C09153=1117.834,-111.203,-46.268,179.703,4.253,148.782
C09154=1117.839,-111.453,-46.260,179.703,4.248,148.781
C09155=1117.844,-111.703,-46.251,179.703,4.243,148.779
C09156=1117.850,-111.953,-46.242,179.703,4.238,148.778
C09157=1117.855,-112.203,-46.234,179.704,4.233,148.777
C09158=1117.861,-112.452,-46.225,179.705,4.228,148.776
C09159=1117.866,-112.702,-46.216,179.705,4.223,148.775
C09160=1117.872,-112.952,-46.207,179.705,4.218,148.773
C09161=1117.877,-113.202,-46.198,179.705,4.213,148.772
C09162=1117.881,-113.417,-46.191,179.706,4.208,148.771
C09163=1117.886,-113.632,-46.183,179.706,4.204,148.770
C09164=1117.890,-113.848,-46.175,179.706,4.199,148.769
C09165=1117.895,-114.063,-46.168,179.706,4.195,148.768
C09166=1117.900,-114.279,-46.161,179.706,4.190,148.767
C09167=1117.905,-114.494,-46.153,179.707,4.186,148.766
C09168=1117.909,-114.710,-46.145,179.707,4.181,148.765
C09169=1117.914,-114.925,-46.137,179.707,4.177,148.764
C09170=1117.919,-115.174,-46.129,179.707,4.171,148.763
C09171=1117.925,-115.424,-46.120,179.708,4.166,148.761
C09172=1117.930,-115.674,-46.112,179.708,4.161,148.760
C09173=1117.936,-115.924,-46.103,179.708,4.156,148.759
C09174=1117.941,-116.174,-46.094,179.709,4.150,148.757
C09175=1117.946,-116.423,-46.086,179.709,4.145,148.756
C09176=1117.952,-116.673,-46.077,179.709,4.139,148.755
C09177=1117.957,-116.923,-46.068,179.709,4.134,148.754
C09178=1117.962,-117.173,-46.060,179.709,4.129,148.753
C09179=1117.968,-117.422,-46.051,179.710,4.124,148.751
C09180=1117.973,-117.672,-46.042,179.710,4.119,148.750
C09181=1117.979,-117.923,-46.034,179.710,4.113,148.749
C09182=1117.984,-118.172,-46.025,179.711,4.108,148.748
C09183=1117.990,-118.422,-46.016,179.711,4.103,148.747
C09184=1117.995,-118.671,-46.008,179.712,4.098,148.745
C09185=1117.999,-118.922,-46.000,179.712,4.092,148.744
C09186=1118.005,-119.171,-45.991,179.712,4.087,148.743
C09187=1118.010,-119.421,-45.983,179.712,4.081,148.742
C09188=1118.016,-119.671,-45.974,179.712,4.076,148.740
C09189=1118.022,-119.920,-45.966,179.712,4.071,148.739
C09190=1118.027,-120.170,-45.957,179.713,4.066,148.738
C09191=1118.032,-120.420,-45.948,179.714,4.060,148.736
C09192=1118.038,-120.670,-45.940,179.714,4.055,148.735
C09193=1118.043,-120.920,-45.931,179.714,4.050,148.734
C09194=1118.049,-121.170,-45.923,179.714,4.045,148.733
C09195=1118.054,-121.419,-45.915,179.714,4.039,148.732
C09196=1118.059,-121.669,-45.906,179.714,4.033,148.730
C09197=1118.064,-121.919,-45.898,179.715,4.028,148.729
C09198=1118.070,-122.168,-45.890,179.715,4.023,148.728
C09199=1118.075,-122.418,-45.881,179.716,4.018,148.727
C09200=1118.081,-122.669,-45.873,179.715,4.012,148.725
C09201=1118.087,-122.918,-45.864,179.716,4.006,148.724
C09202=1118.091,-123.168,-45.856,179.717,4.001,148.723
C09203=1118.097,-123.417,-45.848,179.717,3.996,148.721
C09204=1118.103,-123.668,-45.840,179.717,3.991,148.720
C09205=1118.108,-123.917,-45.831,179.717,3.985,148.719
C09206=1118.114,-124.167,-45.823,179.717,3.979,148.718
C09207=1118.118,-124.417,-45.815,179.718,3.974,148.716
C09208=1118.123,-124.667,-45.806,179.718,3.969,148.715
C09209=1118.129,-124.916,-45.798,179.719,3.963,148.714
C09210=1118.135,-125.166,-45.789,179.718,3.957,148.713
C09211=1118.141,-125.416,-45.781,179.719,3.952,148.711
C09212=1118.145,-125.666,-45.773,179.719,3.947,148.710
C09213=1118.151,-125.915,-45.765,179.720,3.942,148.709
C09214=1118.157,-126.166,-45.757,179.720,3.935,148.707
C09215=1118.162,-126.416,-45.748,179.720,3.930,148.706
C09216=1118.167,-126.665,-45.741,179.721,3.925,148.705
C09217=1118.172,-126.915,-45.732,179.721,3.920,148.704
C09218=1118.177,-127.131,-45.725,179.721,3.914,148.702
C09219=1118.182,-127.345,-45.718,179.721,3.909,148.701
C09220=1118.187,-127.561,-45.711,179.721,3.905,148.700
C09221=1118.191,-127.776,-45.704,179.722,3.900,148.699
C09222=1118.196,-127.992,-45.697,179.722,3.895,148.698
C09223=1118.201,-128.207,-45.690,179.722,3.890,148.697
C09224=1118.205,-128.422,-45.683,179.723,3.886,148.696
C09225=1118.210,-128.639,-45.676,179.723,3.881,148.695
C09226=1117.787,-128.629,-45.702,179.730,3.886,148.693
C09227=1117.782,-128.414,-45.709,179.730,3.890,148.694
C09228=1117.777,-128.198,-45.716,179.729,3.895,148.696
C09229=1117.773,-127.982,-45.724,179.730,3.900,148.697
C09230=1117.768,-127.767,-45.730,179.729,3.904,148.698
C09231=1117.764,-127.551,-45.737,179.729,3.909,148.699
C09232=1117.759,-127.336,-45.744,179.729,3.914,148.700
C09233=1117.754,-127.120,-45.751,179.728,3.918,148.701
C09234=1117.750,-126.906,-45.758,179.728,3.923,148.702
C09235=1117.744,-126.655,-45.766,179.727,3.929,148.704
C09236=1117.738,-126.406,-45.775,179.728,3.935,148.705
C09237=1117.734,-126.156,-45.783,179.727,3.940,148.706
C09238=1117.728,-125.907,-45.791,179.727,3.945,148.707
C09239=1117.722,-125.656,-45.799,179.726,3.951,148.709
C09240=1117.717,-125.406,-45.808,179.726,3.957,148.710
C09241=1117.711,-125.157,-45.816,179.726,3.962,148.711
C09242=1117.707,-124.907,-45.824,179.726,3.967,148.712
C09243=1117.701,-124.657,-45.832,179.725,3.972,148.714
C09244=1117.696,-124.408,-45.841,179.725,3.978,148.715
C09245=1117.690,-124.158,-45.850,179.725,3.984,148.716
C09246=1117.684,-123.908,-45.858,179.725,3.989,148.717
C09247=1117.680,-123.658,-45.866,179.724,3.994,148.719
C09248=1117.674,-123.408,-45.874,179.724,3.999,148.720
C09249=1117.669,-123.159,-45.883,179.724,4.005,148.721
C09250=1117.663,-122.908,-45.891,179.724,4.011,148.723
C09251=1117.657,-122.659,-45.899,179.723,4.016,148.724
C09252=1117.652,-122.409,-45.908,179.722,4.021,148.725
C09253=1117.647,-122.159,-45.917,179.722,4.027,148.726
C09254=1117.642,-121.910,-45.924,179.722,4.032,148.728
C09255=1117.637,-121.660,-45.933,179.722,4.038,148.729
C09256=1117.631,-121.410,-45.942,179.721,4.043,148.730
C09257=1117.625,-121.160,-45.950,179.721,4.048,148.732
C09258=1117.620,-120.911,-45.959,179.721,4.054,148.733
C09259=1117.615,-120.660,-45.967,179.720,4.059,148.734
C09260=1117.610,-120.410,-45.976,179.720,4.064,148.735
C09261=1117.604,-120.161,-45.985,179.720,4.069,148.736
C09262=1117.598,-119.911,-45.993,179.720,4.075,148.738
C09263=1117.593,-119.661,-46.002,179.719,4.081,148.739
C09264=1117.588,-119.412,-46.010,179.719,4.086,148.740
C09265=1117.583,-119.162,-46.018,179.719,4.091,148.741
C09266=1117.577,-118.912,-46.027,179.719,4.096,148.743
C09267=1117.572,-118.663,-46.035,179.718,4.101,148.744
C09268=1117.567,-118.413,-46.044,179.718,4.107,148.745
C09269=1117.561,-118.162,-46.052,179.717,4.112,148.747
C09270=1117.556,-117.912,-46.061,179.717,4.117,148.748
C09271=1117.550,-117.663,-46.070,179.717,4.123,148.749
C09272=1117.545,-117.413,-46.079,179.717,4.128,148.750
C09273=1117.540,-117.164,-46.088,179.717,4.134,148.751
C09274=1117.534,-116.913,-46.096,179.716,4.139,148.753
C09275=1117.529,-116.664,-46.104,179.716,4.144,148.754
C09276=1117.523,-116.414,-46.113,179.716,4.149,148.755
C09277=1117.518,-116.164,-46.122,179.716,4.154,148.756
C09278=1117.513,-115.914,-46.131,179.715,4.159,148.757
C09279=1117.507,-115.665,-46.139,179.715,4.165,148.759
C09280=1117.502,-115.415,-46.148,179.714,4.170,148.760
C09281=1117.497,-115.165,-46.157,179.714,4.175,148.761
C09282=1117.491,-114.915,-46.165,179.714,4.180,148.763
C09283=1117.487,-114.700,-46.173,179.714,4.185,148.763
C09284=1117.482,-114.485,-46.181,179.713,4.190,148.765
C09285=1117.477,-114.270,-46.188,179.713,4.194,148.766
C09286=1117.473,-114.054,-46.196,179.713,4.198,148.767
C09287=1117.468,-113.838,-46.203,179.712,4.203,148.768
C09288=1117.463,-113.623,-46.211,179.713,4.207,148.769
C09289=1117.458,-113.408,-46.218,179.712,4.211,148.770
C09290=1117.454,-113.192,-46.226,179.712,4.217,148.771
C09291=1117.448,-112.943,-46.235,179.712,4.222,148.772
C09292=1117.443,-112.693,-46.244,179.711,4.227,148.773
C09293=1117.438,-112.443,-46.253,179.711,4.232,148.775
C09294=1117.433,-112.194,-46.262,179.711,4.237,148.776
C09295=1117.427,-111.944,-46.270,179.711,4.242,148.777
C09296=1117.422,-111.695,-46.279,179.710,4.248,148.778
C09297=1117.416,-111.445,-46.288,179.710,4.253,148.779
C09298=1117.411,-111.195,-46.297,179.710,4.258,148.781
C09299=1117.405,-110.945,-46.306,179.710,4.263,148.782
C09300=1117.400,-110.695,-46.315,179.709,4.267,148.783
C09301=1117.395,-110.445,-46.324,179.709,4.273,148.784
C09302=1117.390,-110.195,-46.333,179.708,4.278,148.785
C09303=1117.384,-109.946,-46.342,179.708,4.283,148.787
C09304=1117.379,-109.696,-46.350,179.708,4.288,148.788
C09305=1117.374,-109.446,-46.359,179.708,4.293,148.789
C09306=1117.368,-109.196,-46.369,179.707,4.298,148.790
C09307=1117.363,-108.946,-46.378,179.707,4.304,148.791
C09308=1117.358,-108.696,-46.387,179.707,4.309,148.793
C09309=1117.352,-108.447,-46.396,179.707,4.314,148.794
C09310=1117.347,-108.197,-46.404,179.706,4.319,148.795
C09311=1117.341,-107.947,-46.414,179.706,4.324,148.796
C09312=1117.336,-107.698,-46.423,179.706,4.329,148.797
C09313=1117.331,-107.448,-46.432,179.705,4.334,148.799
C09314=1117.326,-107.198,-46.441,179.705,4.339,148.800
C09315=1117.320,-106.948,-46.450,179.704,4.344,148.801
C09316=1117.314,-106.698,-46.459,179.704,4.349,148.802
C09317=1117.309,-106.448,-46.468,179.704,4.354,148.803
C09318=1117.304,-106.199,-46.477,179.704,4.360,148.805
C09319=1117.299,-105.949,-46.486,179.704,4.365,148.806
C09320=1117.293,-105.699,-46.496,179.703,4.370,148.807
C09321=1117.288,-105.449,-46.505,179.703,4.375,148.808
C09322=1117.282,-105.200,-46.514,179.702,4.379,148.809
C09323=1117.277,-104.950,-46.523,179.702,4.385,148.811
C09324=1117.271,-104.700,-46.532,179.702,4.390,148.812
C09325=1117.266,-104.451,-46.542,179.702,4.395,148.813
C09326=1117.261,-104.201,-46.551,179.701,4.400,148.814
C09327=1117.256,-103.951,-46.559,179.701,4.405,148.815
C09328=1117.250,-103.701,-46.569,179.701,4.410,148.817
C09329=1117.245,-103.451,-46.578,179.700,4.415,148.818
C09330=1117.240,-103.202,-46.587,179.700,4.420,148.819
C09331=1117.234,-102.952,-46.597,179.700,4.425,148.820
C09332=1117.229,-102.702,-46.606,179.699,4.430,148.821
C09333=1117.224,-102.452,-46.615,179.699,4.435,148.822
C09334=1117.219,-102.203,-46.624,179.699,4.441,148.824
C09335=1117.213,-101.953,-46.634,179.699,4.445,148.825
C09336=1117.208,-101.703,-46.643,179.698,4.450,148.826
C09337=1117.203,-101.454,-46.652,179.698,4.455,148.827
C09338=1117.197,-101.203,-46.662,179.698,4.460,148.828
C09339=1117.192,-100.988,-46.669,179.697,4.464,148.829
C09340=1117.188,-100.773,-46.677,179.697,4.468,148.830
C09341=1117.184,-100.558,-46.686,179.697,4.473,148.831
C09342=1117.180,-100.342,-46.694,179.697,4.477,148.832
C09343=1117.174,-100.127,-46.702,179.696,4.481,148.833
C09344=1117.169,-99.912,-46.710,179.696,4.485,148.834
C09345=1117.165,-99.697,-46.718,179.696,4.490,148.835
C09346=1117.160,-99.482,-46.726,179.696,4.494,148.836
C09347=1117.156,-99.232,-46.736,179.695,4.499,148.838
C09348=1117.150,-98.982,-46.745,179.695,4.505,148.839
C09349=1117.145,-98.732,-46.754,179.694,4.509,148.840
C09350=1117.139,-98.483,-46.764,179.694,4.514,148.841
C09351=1117.134,-98.233,-46.773,179.694,4.519,148.842
C09352=1117.128,-97.983,-46.783,179.694,4.524,148.843
C09353=1117.123,-97.734,-46.792,179.693,4.529,148.845
C09354=1117.118,-97.484,-46.801,179.693,4.534,148.846
C09355=1117.112,-97.234,-46.811,179.693,4.539,148.847
C09356=1117.107,-96.984,-46.820,179.692,4.544,148.848
C09357=1117.101,-96.735,-46.830,179.692,4.549,148.849
C09358=1117.097,-96.484,-46.840,179.691,4.554,148.851
C09359=1117.091,-96.235,-46.850,179.691,4.559,148.852
C09360=1117.086,-95.985,-46.859,179.691,4.564,148.853
C09361=1117.080,-95.735,-46.868,179.690,4.568,148.854
C09362=1117.075,-95.485,-46.878,179.690,4.574,148.855
C09363=1117.069,-95.235,-46.887,179.690,4.579,148.857
C09364=1117.065,-94.986,-46.897,179.690,4.584,148.858
C09365=1117.059,-94.736,-46.906,179.689,4.588,148.859
C09366=1117.054,-94.487,-46.916,179.689,4.593,148.860
C09367=1117.048,-94.236,-46.926,179.689,4.598,148.861
C09368=1117.043,-93.987,-46.935,179.688,4.603,148.862
C09369=1117.037,-93.737,-46.945,179.687,4.608,148.864
C09370=1117.033,-93.487,-46.955,179.687,4.612,148.865
C09371=1117.027,-93.238,-46.965,179.686,4.617,148.866
C09372=1117.022,-92.988,-46.974,179.686,4.622,148.867
C09373=1117.017,-92.738,-46.984,179.685,4.626,148.868
C09374=1117.011,-92.488,-46.993,179.684,4.632,148.870
C09375=1117.006,-92.239,-47.003,179.683,4.636,148.871
C09376=1117.001,-91.989,-47.012,179.683,4.641,148.872
C09377=1116.995,-91.739,-47.022,179.682,4.646,148.873
C09378=1116.990,-91.489,-47.031,179.682,4.651,148.875
C09379=1116.985,-91.239,-47.042,179.682,4.656,148.876
C09380=1116.980,-90.990,-47.051,179.681,4.661,148.877
C09381=1116.974,-90.740,-47.061,179.680,4.666,148.878
C09382=1116.968,-90.490,-47.071,179.680,4.670,148.880
C09383=1116.963,-90.240,-47.080,179.679,4.675,148.881
C09384=1116.958,-89.991,-47.090,179.679,4.680,148.882
C09385=1116.953,-89.741,-47.100,179.678,4.685,148.883
C09386=1116.948,-89.491,-47.110,179.678,4.690,148.885
C09387=1116.942,-89.241,-47.120,179.677,4.695,148.886
C09388=1116.937,-88.992,-47.129,179.677,4.700,148.887
C09389=1116.931,-88.742,-47.139,179.677,4.705,148.888
C09390=1116.926,-88.493,-47.148,179.676,4.709,148.889
C09391=1116.921,-88.242,-47.159,179.675,4.715,148.891
C09392=1116.915,-87.992,-47.169,179.675,4.720,148.892
C09393=1116.911,-87.743,-47.178,179.674,4.724,148.893
C09394=1116.905,-87.493,-47.188,179.674,4.730,148.894
C09395=1116.901,-87.278,-47.196,179.674,4.734,148.895
C09396=1116.896,-87.063,-47.205,179.673,4.738,148.896
C09397=1116.892,-86.848,-47.214,179.673,4.743,148.897
C09398=1116.887,-86.633,-47.222,179.673,4.747,148.898
C09399=1116.882,-86.417,-47.231,179.672,4.751,148.899
C09400=1116.878,-86.203,-47.239,179.671,4.755,148.901
C09401=1116.874,-85.988,-47.248,179.672,4.760,148.902
C09402=1116.868,-85.772,-47.256,179.671,4.764,148.903
C09403=1116.864,-85.522,-47.266,179.671,4.770,148.904
C09404=1116.858,-85.273,-47.276,179.670,4.774,148.905
C09405=1116.853,-85.023,-47.286,179.670,4.779,148.906
C09406=1116.848,-84.773,-47.295,179.670,4.784,148.907
C09407=1116.842,-84.524,-47.306,179.670,4.789,148.909
C09408=1116.837,-84.273,-47.316,179.669,4.795,148.910
C09409=1116.831,-84.024,-47.326,179.669,4.799,148.911
C09410=1116.827,-83.775,-47.336,179.668,4.804,148.912
C09411=1116.821,-83.524,-47.345,179.668,4.810,148.914
C09412=1116.816,-83.274,-47.356,179.668,4.815,148.915
C09413=1116.811,-83.025,-47.366,179.667,4.820,148.916
C09414=1116.805,-82.775,-47.376,179.667,4.825,148.917
C09415=1116.800,-82.526,-47.386,179.667,4.830,148.918
C09416=1116.795,-82.276,-47.397,179.667,4.835,148.919
C09417=1116.789,-82.026,-47.406,179.666,4.840,148.921
C09418=1116.784,-81.776,-47.416,179.666,4.845,148.922
C09419=1116.779,-81.526,-47.426,179.666,4.850,148.923
C09420=1116.773,-81.277,-47.437,179.666,4.855,148.924
C09421=1116.768,-81.027,-47.446,179.665,4.861,148.926
C09422=1116.763,-80.778,-47.456,179.665,4.866,148.927
C09423=1116.758,-80.527,-47.467,179.665,4.871,148.928
C09424=1116.752,-80.278,-47.477,179.665,4.876,148.929
C09425=1116.747,-80.028,-47.487,179.664,4.881,148.930
C09426=1116.742,-79.778,-47.497,179.664,4.886,148.931
C09427=1116.736,-79.528,-47.507,179.664,4.892,148.933
C09428=1116.731,-79.279,-47.517,179.664,4.897,148.934
C09429=1116.725,-79.029,-47.527,179.664,4.902,148.935
C09430=1116.720,-78.779,-47.538,179.664,4.907,148.936
C09431=1116.715,-78.529,-47.548,179.663,4.912,148.937
C09432=1116.709,-78.280,-47.558,179.663,4.917,148.938
C09433=1116.705,-78.030,-47.568,179.663,4.923,148.940
C09434=1116.699,-77.780,-47.578,179.663,4.928,148.941
C09435=1116.694,-77.531,-47.589,179.663,4.933,148.942
C09436=1116.689,-77.281,-47.599,179.663,4.938,148.943
C09437=1116.683,-77.031,-47.609,179.662,4.943,148.944
C09438=1116.677,-76.782,-47.620,179.662,4.948,148.945
C09439=1116.672,-76.531,-47.630,179.663,4.953,148.946
C09440=1116.667,-76.282,-47.640,179.662,4.958,148.948
C09441=1116.662,-76.032,-47.650,179.663,4.964,148.949
C09442=1116.657,-75.783,-47.661,179.663,4.969,148.950
C09443=1116.652,-75.533,-47.671,179.663,4.974,148.951
C09444=1116.647,-75.283,-47.682,179.662,4.980,148.952
C09445=1116.641,-75.034,-47.692,179.662,4.985,148.953
C09446=1116.635,-74.784,-47.702,179.662,4.990,148.955
C09447=1116.630,-74.534,-47.713,179.662,4.995,148.956
C09448=1116.625,-74.284,-47.723,179.662,5.000,148.957
C09449=1116.620,-74.034,-47.734,179.663,5.006,148.958
C09450=1116.614,-73.784,-47.744,179.663,5.011,148.959
C09451=1116.610,-73.569,-47.753,179.662,5.015,148.960
C09452=1116.605,-73.355,-47.762,179.663,5.020,148.961
C09453=1116.601,-73.140,-47.772,179.663,5.024,148.962
C09454=1116.597,-72.924,-47.780,179.662,5.029,148.963
C09455=1116.592,-72.710,-47.789,179.663,5.034,148.964
C09456=1116.587,-72.494,-47.799,179.663,5.037,148.965
C09457=1116.582,-72.280,-47.807,179.663,5.042,148.966
C09458=1116.578,-72.064,-47.816,179.663,5.047,148.967
C09459=1116.573,-71.815,-47.827,179.663,5.052,148.968
C09460=1116.567,-71.565,-47.838,179.663,5.057,148.969
C09461=1116.562,-71.315,-47.848,179.663,5.062,148.970
C09462=1116.557,-71.065,-47.858,179.663,5.067,148.971
C09463=1116.551,-70.816,-47.869,179.664,5.073,148.972
C09464=1116.547,-70.566,-47.880,179.664,5.078,148.973
C09465=1116.541,-70.317,-47.890,179.664,5.083,148.974
C09466=1116.536,-70.066,-47.901,179.664,5.088,148.975
C09467=1116.531,-69.817,-47.912,179.665,5.094,148.976
C09468=1116.526,-69.567,-47.922,179.665,5.099,148.978
C09469=1116.520,-69.318,-47.932,179.665,5.104,148.979
C09470=1116.514,-69.067,-47.944,179.665,5.109,148.980
C09471=1116.509,-68.818,-47.955,179.665,5.115,148.981
C09472=1116.504,-68.568,-47.965,179.666,5.120,148.982
C09473=1116.498,-68.318,-47.975,179.666,5.125,148.983
C09474=1116.494,-68.069,-47.987,179.666,5.129,148.984
C09475=1116.488,-67.819,-47.997,179.666,5.135,148.985
C09476=1116.483,-67.570,-48.008,179.666,5.141,148.986
C09477=1116.478,-67.320,-48.018,179.667,5.145,148.987
C09478=1116.473,-67.070,-48.029,179.667,5.151,148.988
C09479=1116.467,-66.820,-48.040,179.668,5.156,148.989
C09480=1116.462,-66.570,-48.051,179.667,5.161,148.990
C09481=1116.457,-66.321,-48.062,179.668,5.167,148.991
C09482=1116.452,-66.071,-48.073,179.669,5.171,148.992
C09483=1116.447,-65.821,-48.083,179.669,5.177,148.993
C09484=1116.441,-65.572,-48.094,179.670,5.182,148.994
C09485=1116.436,-65.321,-48.105,179.669,5.187,148.995
C09486=1116.430,-65.072,-48.116,179.670,5.192,148.996
C09487=1116.425,-64.822,-48.127,179.671,5.198,148.997
C09488=1116.420,-64.573,-48.138,179.671,5.203,148.998
C09489=1116.415,-64.323,-48.148,179.671,5.208,148.999
C09490=1116.410,-64.073,-48.160,179.672,5.213,149.000
C09491=1116.404,-63.824,-48.170,179.672,5.218,149.001
C09492=1116.399,-63.574,-48.182,179.673,5.224,149.002
C09493=1116.394,-63.324,-48.192,179.673,5.229,149.003
C09494=1116.389,-63.075,-48.203,179.673,5.234,149.004
C09495=1116.384,-62.825,-48.215,179.674,5.239,149.005
C09496=1116.378,-62.575,-48.225,179.675,5.244,149.006
C09497=1116.373,-62.326,-48.236,179.675,5.249,149.007
C09498=1116.368,-62.075,-48.247,179.676,5.254,149.008
C09499=1116.362,-61.826,-48.259,179.676,5.259,149.009
C09500=1116.358,-61.577,-48.270,179.677,5.265,149.010
C09501=1116.352,-61.327,-48.280,179.677,5.270,149.011
C09502=1116.346,-61.077,-48.292,179.678,5.275,149.012
C09503=1116.341,-60.827,-48.303,179.679,5.280,149.013
C09504=1116.336,-60.578,-48.313,179.679,5.285,149.014
C09505=1116.331,-60.328,-48.325,179.680,5.290,149.015
C09506=1116.326,-60.078,-48.337,179.680,5.295,149.016
C09507=1116.321,-59.863,-48.346,179.680,5.299,149.017
C09508=1116.317,-59.649,-48.356,179.680,5.303,149.018
C09509=1116.312,-59.433,-48.365,179.680,5.307,149.018
C09510=1116.308,-59.218,-48.375,179.680,5.312,149.019
C09511=1116.304,-59.004,-48.384,179.680,5.316,149.020
C09512=1116.299,-58.788,-48.394,179.680,5.320,149.021
C09513=1116.295,-58.573,-48.404,179.680,5.324,149.022
C09514=1116.290,-58.358,-48.413,179.679,5.328,149.023
C09515=1116.284,-58.109,-48.424,179.679,5.333,149.024
C09516=1116.280,-57.859,-48.436,179.679,5.337,149.025
C09517=1116.275,-57.609,-48.447,179.679,5.342,149.026
C09518=1116.269,-57.360,-48.458,179.679,5.346,149.027
C09519=1116.264,-57.110,-48.469,179.679,5.351,149.028
C09520=1116.258,-56.860,-48.481,179.679,5.356,149.030
C09521=1116.254,-56.610,-48.492,179.678,5.360,149.030
C09522=1116.248,-56.361,-48.503,179.678,5.365,149.032
C09523=1116.243,-56.111,-48.514,179.678,5.369,149.033
C09524=1116.238,-55.861,-48.526,179.678,5.374,149.034
C09525=1116.233,-55.611,-48.537,179.678,5.379,149.035
C09526=1116.227,-55.362,-48.548,179.677,5.384,149.036
C09527=1116.223,-55.113,-48.560,179.678,5.388,149.037
C09528=1116.217,-54.863,-48.572,179.677,5.393,149.038
C09529=1116.212,-54.613,-48.582,179.677,5.398,149.039
C09530=1116.206,-54.363,-48.594,179.677,5.403,149.040
C09531=1116.201,-54.114,-48.605,179.677,5.407,149.041
C09532=1116.196,-53.864,-48.617,179.677,5.412,149.042
C09533=1116.191,-53.614,-48.628,179.676,5.416,149.043
C09534=1116.185,-53.365,-48.640,179.676,5.421,149.044
C09535=1116.181,-53.115,-48.651,179.677,5.426,149.045
C09536=1116.175,-52.865,-48.663,179.676,5.430,149.047
C09537=1116.170,-52.615,-48.673,179.676,5.435,149.048
C09538=1116.164,-52.366,-48.685,179.675,5.440,149.049
C09539=1116.159,-52.116,-48.696,179.676,5.445,149.050
C09540=1116.154,-51.866,-48.708,179.676,5.450,149.051
C09541=1116.149,-51.617,-48.719,179.675,5.454,149.052
C09542=1116.144,-51.367,-48.731,179.675,5.459,149.053
C09543=1116.139,-51.118,-48.742,179.675,5.463,149.054
C09544=1116.133,-50.868,-48.754,179.674,5.468,149.055
C09545=1116.128,-50.618,-48.765,179.675,5.473,149.056
C09546=1116.123,-50.368,-48.777,179.674,5.477,149.057
C09547=1116.118,-50.119,-48.789,179.674,5.482,149.058
C09548=1116.113,-49.869,-48.800,179.675,5.487,149.059
C09549=1116.107,-49.620,-48.812,179.674,5.492,149.061
C09550=1116.102,-49.370,-48.823,179.674,5.497,149.062
C09551=1116.097,-49.120,-48.835,179.673,5.501,149.063
C09552=1116.092,-48.870,-48.846,179.674,5.506,149.064
C09553=1116.087,-48.620,-48.858,179.673,5.511,149.065
C09554=1116.081,-48.372,-48.869,179.673,5.515,149.066
C09555=1116.076,-48.122,-48.881,179.673,5.520,149.067
C09556=1116.071,-47.872,-48.893,179.673,5.524,149.068
C09557=1116.066,-47.622,-48.904,179.673,5.529,149.069
C09558=1116.060,-47.372,-48.916,179.673,5.534,149.070
C09559=1116.056,-47.122,-48.927,179.672,5.539,149.071
C09560=1116.050,-46.873,-48.939,179.672,5.544,149.072
C09561=1116.044,-46.623,-48.951,179.672,5.548,149.074
C09562=1116.040,-46.374,-48.962,179.672,5.553,149.075
C09563=1116.034,-46.158,-48.973,179.672,5.557,149.075
C09564=1116.030,-45.944,-48.983,179.672,5.561,149.076
C09565=1116.026,-45.729,-48.993,179.671,5.565,149.078
C09566=1116.021,-45.514,-49.003,179.671,5.569,149.078
C09567=1116.017,-45.299,-49.013,179.671,5.574,149.079
C09568=1116.013,-45.084,-49.023,179.671,5.578,149.080
C09569=1116.008,-44.869,-49.033,179.671,5.582,149.081
C09570=1116.004,-44.655,-49.044,179.671,5.585,149.082
C09571=1115.999,-44.405,-49.055,179.670,5.590,149.083
C09572=1115.994,-44.155,-49.067,179.670,5.595,149.084
C09573=1115.988,-43.905,-49.079,179.670,5.600,149.085
C09574=1115.983,-43.656,-49.090,179.670,5.604,149.086
C09575=1115.978,-43.406,-49.102,179.670,5.609,149.088
C09576=1115.973,-43.156,-49.115,179.670,5.613,149.088
C09577=1115.968,-42.907,-49.126,179.669,5.618,149.090
C09578=1115.962,-42.658,-49.138,179.671,5.624,149.091
C09579=1115.957,-42.408,-49.150,179.672,5.629,149.091
C09580=1115.951,-42.158,-49.162,179.673,5.634,149.092
C09581=1115.947,-41.909,-49.174,179.674,5.640,149.093
C09582=1115.941,-41.659,-49.185,179.675,5.646,149.094
C09583=1115.936,-41.409,-49.197,179.676,5.650,149.095
C09584=1115.931,-41.159,-49.209,179.677,5.655,149.095
C09585=1115.926,-40.910,-49.221,179.678,5.661,149.096
C09586=1115.921,-40.660,-49.233,179.679,5.667,149.097
C09587=1115.915,-40.410,-49.245,179.680,5.671,149.098
C09588=1115.910,-40.161,-49.258,179.681,5.676,149.099
C09589=1115.905,-39.911,-49.269,179.682,5.681,149.100
C09590=1115.900,-39.661,-49.281,179.683,5.686,149.100
C09591=1115.895,-39.412,-49.293,179.684,5.691,149.101
C09592=1115.890,-39.162,-49.305,179.685,5.697,149.102
C09593=1115.884,-38.912,-49.318,179.685,5.701,149.103
C09594=1115.879,-38.663,-49.330,179.687,5.707,149.104
C09595=1115.874,-38.413,-49.342,179.687,5.711,149.105
C09596=1115.868,-38.163,-49.354,179.687,5.716,149.106
C09597=1115.864,-37.914,-49.365,179.688,5.720,149.106
C09598=1115.859,-37.664,-49.378,179.689,5.726,149.107
C09599=1115.853,-37.414,-49.390,179.690,5.731,149.108
C09600=1115.848,-37.165,-49.403,179.691,5.735,149.109
C09601=1115.843,-36.915,-49.414,179.691,5.740,149.110
C09602=1115.837,-36.665,-49.426,179.692,5.744,149.111
C09603=1115.832,-36.416,-49.439,179.693,5.749,149.111
C09604=1115.827,-36.166,-49.451,179.693,5.754,149.112
C09605=1115.822,-35.917,-49.463,179.694,5.758,149.113
C09606=1115.816,-35.667,-49.475,179.694,5.763,149.114
C09607=1115.812,-35.417,-49.488,179.695,5.767,149.115
C09608=1115.807,-35.168,-49.500,179.695,5.772,149.116
C09609=1115.802,-34.918,-49.512,179.696,5.777,149.117
C09610=1115.797,-34.668,-49.525,179.696,5.782,149.117
C09611=1115.791,-34.418,-49.537,179.697,5.786,149.118
C09612=1115.786,-34.169,-49.549,179.698,5.791,149.119
C09613=1115.781,-33.919,-49.561,179.698,5.795,149.120
C09614=1115.776,-33.670,-49.574,179.698,5.799,149.121
C09615=1115.770,-33.421,-49.586,179.698,5.804,149.122
C09616=1115.765,-33.171,-49.598,179.699,5.809,149.123
C09617=1115.760,-32.921,-49.611,179.699,5.812,149.123
C09618=1115.755,-32.671,-49.623,179.700,5.817,149.124
C09619=1115.750,-32.456,-49.634,179.700,5.821,149.125
C09620=1115.746,-32.241,-49.644,179.700,5.825,149.126
C09621=1115.741,-32.027,-49.656,179.700,5.829,149.127
C09622=1115.737,-31.812,-49.666,179.700,5.832,149.127
C09623=1115.732,-31.597,-49.677,179.700,5.836,149.128
C09624=1115.728,-31.382,-49.687,179.700,5.840,149.129
C09625=1115.724,-31.167,-49.699,179.701,5.844,149.130
C09626=1115.719,-30.952,-49.709,179.701,5.847,149.131
C09627=1115.714,-30.703,-49.721,179.701,5.852,149.131
C09628=1115.709,-30.454,-49.734,179.701,5.856,149.132
C09629=1115.704,-30.204,-49.746,179.701,5.861,149.133
C09630=1115.699,-29.954,-49.759,179.701,5.865,149.134
C09631=1115.694,-29.704,-49.771,179.701,5.869,149.135
C09632=1115.689,-29.455,-49.784,179.701,5.874,149.136
C09633=1115.683,-29.205,-49.796,179.701,5.878,149.137
C09634=1115.677,-28.956,-49.809,179.701,5.881,149.138
C09635=1115.672,-28.706,-49.822,179.701,5.887,149.139
C09636=1115.668,-28.456,-49.835,179.701,5.891,149.140
C09637=1115.662,-28.206,-49.846,179.700,5.894,149.141
C09638=1115.657,-27.957,-49.859,179.700,5.899,149.142
C09639=1115.652,-27.708,-49.872,179.700,5.904,149.143
C09640=1115.647,-27.458,-49.884,179.700,5.908,149.144
C09641=1115.642,-27.208,-49.897,179.700,5.912,149.145
C09642=1115.637,-26.958,-49.909,179.699,5.916,149.146
C09643=1115.632,-26.709,-49.922,179.698,5.920,149.147
C09644=1115.626,-26.459,-49.935,179.698,5.924,149.148
C09645=1115.622,-26.209,-49.948,179.698,5.929,149.149
C09646=1115.616,-25.960,-49.961,179.697,5.933,149.150
C09647=1115.611,-25.710,-49.972,179.697,5.938,149.151
C09648=1115.606,-25.461,-49.985,179.698,5.942,149.152
C09649=1115.601,-25.212,-49.998,179.698,5.947,149.153
C09650=1115.596,-24.961,-50.011,179.699,5.952,149.154
C09651=1115.590,-24.712,-50.024,179.699,5.957,149.155
C09652=1115.585,-24.463,-50.036,179.700,5.961,149.156
C09653=1115.580,-24.213,-50.048,179.700,5.966,149.157
C09654=1115.575,-23.963,-50.061,179.701,5.972,149.158
C09655=1115.570,-23.713,-50.074,179.702,5.976,149.159
C09656=1115.564,-23.464,-50.087,179.702,5.981,149.159
C09657=1115.559,-23.214,-50.100,179.703,5.986,149.160
C09658=1115.555,-22.964,-50.113,179.703,5.991,149.161
C09659=1115.550,-22.715,-50.125,179.704,5.995,149.162
C09660=1115.544,-22.465,-50.138,179.704,6.000,149.163
C09661=1115.539,-22.216,-50.151,179.705,6.005,149.164
C09662=1115.534,-21.966,-50.164,179.705,6.010,149.165
C09663=1115.529,-21.717,-50.177,179.706,6.014,149.166
C09664=1115.523,-21.467,-50.190,179.706,6.019,149.167
C09665=1115.519,-21.217,-50.203,179.707,6.024,149.168
C09666=1115.513,-20.968,-50.215,179.707,6.028,149.168
C09667=1115.508,-20.718,-50.228,179.708,6.033,149.169
C09668=1115.503,-20.468,-50.241,179.709,6.038,149.170
C09669=1115.498,-20.219,-50.254,179.709,6.042,149.171
C09670=1115.493,-19.969,-50.267,179.709,6.047,149.172
C09671=1115.488,-19.719,-50.280,179.710,6.052,149.173
C09672=1115.482,-19.470,-50.293,179.710,6.056,149.174
C09673=1115.477,-19.220,-50.305,179.711,6.061,149.174
C09674=1115.472,-18.970,-50.319,179.711,6.066,149.175
C09675=1115.468,-18.756,-50.330,179.712,6.070,149.176
C09676=1115.463,-18.541,-50.341,179.713,6.074,149.177
C09677=1115.458,-18.327,-50.352,179.713,6.079,149.178
C09678=1115.454,-18.112,-50.364,179.714,6.082,149.178
C09679=1115.450,-17.897,-50.375,179.715,6.086,149.179
C09680=1115.445,-17.683,-50.386,179.715,6.090,149.180
C09681=1115.441,-17.467,-50.398,179.715,6.095,149.181
C09682=1115.437,-17.253,-50.409,179.716,6.098,149.181
C09683=1115.431,-17.004,-50.422,179.716,6.103,149.182
C09684=1115.427,-16.754,-50.435,179.717,6.108,149.183
C09685=1115.421,-16.504,-50.448,179.717,6.112,149.184
C09686=1115.416,-16.255,-50.460,179.718,6.117,149.185
C09687=1115.411,-16.005,-50.475,179.719,6.121,149.185
C09688=1115.406,-15.756,-50.487,179.719,6.126,149.186
C09689=1115.401,-15.506,-50.500,179.720,6.131,149.187
C09690=1115.395,-15.256,-50.513,179.721,6.135,149.188
C09691=1115.390,-15.007,-50.526,179.721,6.140,149.189
C09692=1115.385,-14.757,-50.540,179.722,6.145,149.190
C09693=1115.380,-14.508,-50.553,179.722,6.149,149.191
C09694=1115.375,-14.257,-50.567,179.723,6.154,149.191
C09695=1115.370,-14.008,-50.579,179.724,6.159,149.192
C09696=1115.366,-13.759,-50.593,179.724,6.163,149.193
C09697=1115.360,-13.509,-50.606,179.725,6.168,149.194
C09698=1115.355,-13.259,-50.619,179.725,6.173,149.195
C09699=1115.350,-13.010,-50.633,179.726,6.176,149.195
C09700=1115.345,-12.761,-50.645,179.726,6.181,149.196
C09701=1115.339,-12.510,-50.659,179.727,6.186,149.197
C09702=1115.334,-12.262,-50.672,179.727,6.190,149.198
C09703=1115.329,-12.011,-50.686,179.728,6.195,149.199
C09704=1115.324,-11.762,-50.699,179.729,6.200,149.200
C09705=1115.319,-11.512,-50.713,179.729,6.204,149.201
C09706=1115.313,-11.263,-50.726,179.730,6.209,149.202
C09707=1115.309,-11.013,-50.740,179.731,6.213,149.202
C09708=1115.303,-10.764,-50.753,179.731,6.218,149.203
C09709=1115.299,-10.514,-50.766,179.732,6.223,149.204
C09710=1115.293,-10.265,-50.780,179.733,6.227,149.205
C09711=1115.289,-10.015,-50.793,179.733,6.232,149.206
C09712=1115.283,-9.766,-50.807,179.734,6.237,149.206
C09713=1115.279,-9.515,-50.820,179.734,6.241,149.207
C09714=1115.273,-9.266,-50.833,179.734,6.245,149.208
C09715=1115.268,-9.016,-50.847,179.735,6.250,149.209
C09716=1115.263,-8.766,-50.860,179.735,6.254,149.210
C09717=1115.258,-8.517,-50.874,179.736,6.259,149.210
C09718=1115.253,-8.267,-50.887,179.737,6.263,149.211
C09719=1115.248,-8.018,-50.901,179.737,6.268,149.212
C09720=1115.242,-7.768,-50.914,179.738,6.273,149.213
C09721=1115.237,-7.519,-50.928,179.739,6.277,149.214
C09722=1115.233,-7.269,-50.942,179.739,6.282,149.215
C09723=1115.227,-7.020,-50.955,179.740,6.287,149.216
C09724=1115.222,-6.770,-50.969,179.741,6.291,149.216
C09725=1115.217,-6.521,-50.982,179.741,6.295,149.217
C09726=1115.212,-6.271,-50.996,179.741,6.300,149.218
C09727=1115.207,-6.021,-51.009,179.742,6.304,149.219
C09728=1115.202,-5.772,-51.023,179.743,6.309,149.220
C09729=1115.197,-5.522,-51.037,179.743,6.313,149.220
C09730=1115.191,-5.273,-51.050,179.744,6.318,149.221
C09731=1115.185,-4.912,-51.070,179.745,6.325,149.222
C09732=1115.177,-4.552,-51.089,179.746,6.331,149.224
C09733=1115.170,-4.191,-51.110,179.747,6.338,149.225
C09734=1115.162,-3.831,-51.130,179.748,6.344,149.226
C09735=1115.157,-3.581,-51.144,179.748,6.348,149.227
C09736=1115.152,-3.332,-51.157,179.749,6.353,149.228
C09737=1115.147,-3.082,-51.171,179.749,6.357,149.228
C09738=1115.142,-2.832,-51.185,179.750,6.362,149.229
C09739=1115.137,-2.583,-51.198,179.751,6.366,149.230
C09740=1115.132,-2.333,-51.212,179.751,6.371,149.231
C09741=1115.127,-2.083,-51.227,179.752,6.376,149.232
C09742=1115.121,-1.834,-51.240,179.752,6.381,149.233
C09743=1115.114,-1.516,-51.258,179.754,6.386,149.234
C09744=1115.109,-1.197,-51.275,179.754,6.392,149.235
C09745=1115.102,-0.879,-51.293,179.755,6.398,149.236
C09746=1115.095,-0.561,-51.311,179.755,6.403,149.237
C09747=1115.090,-0.311,-51.325,179.756,6.407,149.238
C09748=1115.085,-0.062,-51.339,179.756,6.412,149.238
C09749=1115.080,0.188,-51.353,179.757,6.417,149.239
C09750=1115.075,0.438,-51.366,179.757,6.421,149.240
C09751=1115.070,0.687,-51.380,179.758,6.426,149.241
C09752=1115.065,0.937,-51.394,179.759,6.431,149.242
C09753=1115.060,1.186,-51.409,179.760,6.435,149.243
C09754=1115.055,1.436,-51.423,179.761,6.440,149.243
C09755=1115.049,1.685,-51.437,179.760,6.443,149.244
C09756=1115.044,1.935,-51.451,179.761,6.448,149.245
C09757=1115.039,2.185,-51.465,179.762,6.453,149.246
C09758=1115.034,2.434,-51.478,179.763,6.457,149.247
C09759=1115.029,2.683,-51.492,179.763,6.462,149.247
C09760=1115.024,2.933,-51.507,179.764,6.467,149.248
C09761=1115.019,3.183,-51.521,179.764,6.471,149.249
C09762=1115.014,3.432,-51.535,179.765,6.476,149.250
C09763=1115.009,3.682,-51.549,179.766,6.480,149.251
C09764=1115.004,3.931,-51.563,179.766,6.484,149.252
C09765=1114.999,4.181,-51.578,179.766,6.489,149.253
C09766=1114.993,4.430,-51.591,179.767,6.494,149.253
C09767=1114.989,4.680,-51.606,179.768,6.498,149.254
C09768=1114.984,4.929,-51.620,179.768,6.503,149.255
C09769=1114.979,5.179,-51.634,179.769,6.508,149.256
C09770=1114.974,5.429,-51.649,179.769,6.512,149.257
C09771=1114.968,5.678,-51.662,179.770,6.517,149.258
C09772=1114.963,5.928,-51.677,179.771,6.521,149.258
C09773=1114.958,6.177,-51.691,179.771,6.526,149.259
C09774=1114.953,6.427,-51.705,179.771,6.530,149.260
C09775=1114.948,6.677,-51.720,179.772,6.535,149.261
C09776=1114.943,6.926,-51.733,179.772,6.539,149.262
C09777=1114.938,7.175,-51.748,179.773,6.544,149.263
C09778=1114.933,7.425,-51.762,179.774,6.548,149.263
C09779=1114.928,7.675,-51.776,179.775,6.553,149.264
C09780=1114.923,7.925,-51.791,179.775,6.558,149.265
C09781=1114.918,8.173,-51.805,179.776,6.563,149.266
C09782=1114.913,8.423,-51.820,179.776,6.567,149.267
C09783=1114.909,8.637,-51.832,179.777,6.571,149.268
C09784=1114.904,8.853,-51.844,179.777,6.575,149.268
C09785=1114.899,9.067,-51.856,179.778,6.579,149.269
C09786=1114.896,9.281,-51.869,179.778,6.583,149.270
C09787=1114.890,9.496,-51.881,179.779,6.587,149.270
C09788=1114.887,9.710,-51.894,179.779,6.591,149.271
C09789=1114.883,9.925,-51.906,179.779,6.594,149.272
C09790=1114.877,10.139,-51.919,179.780,6.599,149.273
C09791=1114.873,10.389,-51.933,179.781,6.603,149.274
C09792=1114.868,10.639,-51.947,179.781,6.608,149.274
C09793=1114.863,10.888,-51.961,179.782,6.613,149.275
C09794=1114.858,11.137,-51.976,179.782,6.616,149.276
C09795=1114.853,11.387,-51.991,179.783,6.621,149.277
C09796=1114.848,11.637,-52.005,179.784,6.626,149.278
C09797=1114.843,11.887,-52.019,179.785,6.630,149.278
C09798=1114.837,12.135,-52.035,179.785,6.635,149.279
C09799=1114.832,12.385,-52.049,179.786,6.639,149.280
C09800=1114.827,12.635,-52.063,179.786,6.644,149.281
C09801=1114.823,12.884,-52.078,179.787,6.649,149.282
C09802=1114.818,13.133,-52.092,179.788,6.653,149.283
C09803=1114.812,13.384,-52.107,179.788,6.658,149.283
C09804=1114.807,13.633,-52.122,179.789,6.662,149.284
C09805=1114.802,13.882,-52.137,179.790,6.667,149.285
C09806=1114.797,14.132,-52.151,179.790,6.671,149.286
C09807=1114.793,14.381,-52.166,179.791,6.675,149.287
C09808=1114.787,14.631,-52.181,179.791,6.680,149.287
C09809=1114.782,14.881,-52.195,179.793,6.684,149.288
C09810=1114.777,15.130,-52.210,179.793,6.689,149.289
C09811=1114.772,15.380,-52.224,179.794,6.694,149.290
C09812=1114.767,15.630,-52.239,179.795,6.698,149.291
C09813=1114.762,15.879,-52.254,179.795,6.703,149.291
C09814=1114.757,16.128,-52.268,179.796,6.707,149.292
C09815=1114.752,16.377,-52.283,179.797,6.712,149.293
C09816=1114.746,16.627,-52.298,179.797,6.716,149.294
C09817=1114.742,16.876,-52.313,179.798,6.720,149.294
C09818=1114.737,17.126,-52.327,179.798,6.725,149.295
C09819=1114.732,17.375,-52.341,179.799,6.729,149.296
C09820=1114.726,17.625,-52.357,179.800,6.734,149.297
C09821=1114.721,17.875,-52.371,179.801,6.738,149.298
C09822=1114.717,18.124,-52.386,179.802,6.743,149.298
C09823=1114.711,18.374,-52.401,179.803,6.747,149.299
C09824=1114.706,18.623,-52.416,179.803,6.752,149.300
C09825=1114.702,18.873,-52.431,179.804,6.755,149.301
C09826=1114.697,19.123,-52.446,179.804,6.760,149.301
C09827=1114.692,19.372,-52.461,179.805,6.764,149.302
C09828=1114.687,19.621,-52.476,179.806,6.769,149.303
C09829=1114.682,19.871,-52.491,179.807,6.773,149.304
C09830=1114.677,20.120,-52.505,179.808,6.778,149.304
C09831=1114.671,20.370,-52.521,179.808,6.782,149.305
C09832=1114.666,20.620,-52.535,179.809,6.787,149.306
C09833=1114.662,20.869,-52.550,179.810,6.791,149.307
C09834=1114.656,21.118,-52.566,179.810,6.795,149.307
C09835=1114.651,21.368,-52.580,179.812,6.799,149.308
C09836=1114.646,21.617,-52.596,179.812,6.804,149.309
C09837=1114.641,21.866,-52.611,179.813,6.808,149.310
C09838=1114.636,22.116,-52.625,179.814,6.813,149.310
C09839=1114.632,22.330,-52.639,179.814,6.816,149.311
C09840=1114.627,22.545,-52.652,179.816,6.820,149.312
C09841=1114.624,22.760,-52.664,179.816,6.824,149.312
C09842=1114.619,22.974,-52.677,179.817,6.827,149.313
C09843=1114.615,23.188,-52.690,179.818,6.832,149.314
C09844=1114.610,23.403,-52.703,179.818,6.835,149.314
C09845=1114.606,23.617,-52.717,179.818,6.839,149.315
C09846=1114.602,23.832,-52.729,179.819,6.843,149.316
C09847=1114.597,24.081,-52.745,179.820,6.847,149.316
C09848=1114.592,24.331,-52.760,179.821,6.851,149.317
C09849=1114.586,24.581,-52.774,179.822,6.855,149.317
C09850=1114.582,24.830,-52.789,179.823,6.860,149.318
C09851=1114.576,25.079,-52.805,179.824,6.864,149.319
C09852=1114.572,25.328,-52.820,179.825,6.869,149.320
C09853=1114.567,25.578,-52.836,179.825,6.873,149.321
C09854=1114.562,25.828,-52.850,179.826,6.877,149.321
C09855=1114.556,26.077,-52.866,179.827,6.881,149.322
C09856=1114.552,26.326,-52.881,179.828,6.885,149.323
C09857=1114.546,26.576,-52.896,179.828,6.890,149.323
C09858=1114.541,26.825,-52.912,179.829,6.894,149.324
C09859=1114.537,27.076,-52.927,179.830,6.899,149.325
C09860=1114.531,27.325,-52.942,179.832,6.903,149.325
C09861=1114.527,27.574,-52.957,179.832,6.907,149.326
C09862=1114.521,27.824,-52.973,179.833,6.911,149.327
C09863=1114.517,28.073,-52.988,179.834,6.916,149.328
C09864=1114.512,28.323,-53.004,179.835,6.920,149.328
C09865=1114.506,28.572,-53.019,179.836,6.924,149.329
C09866=1114.502,28.821,-53.034,179.837,6.929,149.329
C09867=1114.496,29.071,-53.050,179.838,6.933,149.330
C09868=1114.491,29.320,-53.066,179.838,6.937,149.331
C09869=1114.487,29.570,-53.080,179.839,6.941,149.332
C09870=1114.481,29.820,-53.096,179.840,6.945,149.332
C09871=1114.477,30.069,-53.111,179.841,6.950,149.333
C09872=1114.471,30.318,-53.126,179.842,6.954,149.334
C09873=1114.466,30.568,-53.142,179.843,6.958,149.334
C09874=1114.462,30.818,-53.157,179.844,6.963,149.335
C09875=1114.456,31.067,-53.173,179.845,6.966,149.336
C09876=1114.451,31.316,-53.188,179.846,6.970,149.336
C09877=1114.446,31.565,-53.203,179.846,6.975,149.337
C09878=1114.442,31.816,-53.219,179.847,6.979,149.338
C09879=1114.436,32.065,-53.235,179.848,6.984,149.338
C09880=1114.431,32.314,-53.251,179.849,6.988,149.339
C09881=1114.427,32.564,-53.267,179.850,6.992,149.340
C09882=1114.422,32.813,-53.282,179.851,6.996,149.340
C09883=1114.416,33.062,-53.298,179.852,7.000,149.341
C09884=1114.412,33.311,-53.313,179.853,7.005,149.342
C09885=1114.407,33.562,-53.329,179.854,7.009,149.342
C09886=1114.402,33.811,-53.344,179.855,7.013,149.343
C09887=1114.396,34.060,-53.360,179.856,7.017,149.344
C09888=1114.392,34.310,-53.375,179.857,7.021,149.344
C09889=1114.387,34.560,-53.391,179.858,7.025,149.345
C09890=1114.382,34.808,-53.407,179.859,7.030,149.346
C09891=1114.376,35.058,-53.423,179.860,7.034,149.346
C09892=1114.371,35.308,-53.439,179.861,7.038,149.347
C09893=1114.367,35.557,-53.454,179.862,7.043,149.348
C09894=1114.361,35.806,-53.469,179.862,7.046,149.348
C09895=1114.357,36.021,-53.483,179.864,7.050,149.349
C09896=1114.353,36.235,-53.497,179.864,7.053,149.349
C09897=1114.349,36.449,-53.510,179.865,7.057,149.350
C09898=1114.344,36.664,-53.524,179.866,7.061,149.350
C09899=1114.340,36.878,-53.538,179.867,7.064,149.351
C09900=1114.335,37.093,-53.551,179.868,7.068,149.352
C09901=1114.331,37.307,-53.565,179.868,7.071,149.352
C09902=1114.327,37.522,-53.578,179.870,7.075,149.353
C09903=1114.322,37.771,-53.595,179.871,7.079,149.353
C09904=1114.318,38.020,-53.610,179.871,7.083,149.354
C09905=1114.312,38.270,-53.626,179.872,7.087,149.355
C09906=1114.307,38.520,-53.641,179.873,7.091,149.355
C09907=1114.302,38.768,-53.658,179.875,7.096,149.356
C09908=1114.298,39.019,-53.674,179.876,7.100,149.357
C09909=1114.292,39.268,-53.689,179.877,7.104,149.357
C09910=1114.287,39.517,-53.706,179.878,7.108,149.358
C09911=1114.282,39.767,-53.722,179.879,7.112,149.358
C09912=1114.277,40.016,-53.737,179.880,7.116,149.359
C09913=1114.272,40.266,-53.754,179.881,7.120,149.360
C09914=1114.268,40.515,-53.769,179.882,7.125,149.360
C09915=1114.263,40.764,-53.785,179.883,7.129,149.361
C09916=1114.258,41.014,-53.801,179.884,7.133,149.361
C09917=1114.253,41.263,-53.817,179.885,7.136,149.362
C09918=1114.248,41.513,-53.833,179.886,7.141,149.363
C09919=1114.243,41.762,-53.849,179.887,7.145,149.363
C09920=1114.238,42.011,-53.866,179.888,7.149,149.364
C09921=1114.233,42.261,-53.881,179.890,7.153,149.364
C09922=1114.228,42.510,-53.897,179.891,7.158,149.365
C09923=1114.223,42.760,-53.913,179.891,7.161,149.366
C09924=1114.218,43.009,-53.930,179.892,7.165,149.366
C09925=1114.213,43.259,-53.946,179.893,7.170,149.367
C09926=1114.208,43.507,-53.962,179.895,7.174,149.367
C09927=1114.203,43.758,-53.978,179.896,7.178,149.368
C09928=1114.198,44.006,-53.994,179.897,7.182,149.369
C09929=1114.193,44.256,-54.010,179.898,7.186,149.369
C09930=1114.188,44.505,-54.027,179.899,7.190,149.370
C09931=1114.183,44.755,-54.042,179.900,7.194,149.370
C09932=1114.178,45.004,-54.059,179.901,7.198,149.371
C09933=1114.173,45.254,-54.075,179.902,7.203,149.372
C09934=1114.168,45.503,-54.092,179.904,7.207,149.372
C09935=1114.163,45.753,-54.108,179.904,7.210,149.373
C09936=1114.158,46.002,-54.124,179.905,7.214,149.373
C09937=1114.153,46.252,-54.141,179.906,7.219,149.374
C09938=1114.148,46.501,-54.156,179.908,7.223,149.375
C09939=1114.144,46.751,-54.173,179.909,7.227,149.375
C09940=1114.139,47.000,-54.189,179.910,7.231,149.376
C09941=1114.134,47.249,-54.205,179.911,7.234,149.376
C09942=1114.129,47.499,-54.222,179.912,7.239,149.377
C09943=1114.123,47.748,-54.239,179.913,7.243,149.378
C09944=1114.119,47.998,-54.255,179.915,7.247,149.378
C09945=1114.114,48.247,-54.271,179.916,7.251,149.379
C09946=1114.109,48.496,-54.288,179.917,7.255,149.379
C09947=1114.105,48.746,-54.304,179.918,7.259,149.380
C09948=1114.099,48.995,-54.320,179.919,7.263,149.380
C09949=1114.094,49.245,-54.337,179.920,7.267,149.381
C09950=1114.089,49.494,-54.353,179.922,7.271,149.381
C09951=1114.085,49.708,-54.367,179.922,7.275,149.382
C09952=1114.081,49.923,-54.381,179.924,7.278,149.383
C09953=1114.077,50.137,-54.396,179.925,7.282,149.383
C09954=1114.072,50.352,-54.410,179.926,7.285,149.383
C09955=1114.068,50.565,-54.424,179.926,7.288,149.384
C09956=1114.064,50.780,-54.438,179.928,7.292,149.384
C09957=1114.059,50.994,-54.452,179.928,7.295,149.385
C09958=1114.056,51.208,-54.467,179.929,7.298,149.385
C09959=1114.050,51.457,-54.483,179.931,7.303,149.386
C09960=1114.045,51.707,-54.499,179.932,7.307,149.387
C09961=1114.041,51.957,-54.516,179.933,7.311,149.387
C09962=1114.035,52.206,-54.533,179.934,7.315,149.388
C09963=1114.031,52.456,-54.550,179.936,7.319,149.388
C09964=1114.025,52.704,-54.566,179.936,7.323,149.389
C09965=1114.021,52.954,-54.583,179.938,7.327,149.389
C09966=1114.016,53.204,-54.600,179.939,7.331,149.390
C09967=1114.011,53.452,-54.616,179.940,7.335,149.391
C09968=1114.006,53.702,-54.633,179.942,7.339,149.391
C09969=1114.001,53.952,-54.649,179.943,7.343,149.392
C09970=1113.996,54.201,-54.666,179.944,7.347,149.392
C09971=1113.991,54.451,-54.682,179.945,7.351,149.393
C09972=1113.986,54.700,-54.700,179.946,7.355,149.393
C09973=1113.981,54.949,-54.716,179.947,7.359,149.394
C09974=1113.976,55.199,-54.733,179.949,7.363,149.394
C09975=1113.971,55.448,-54.750,179.950,7.367,149.395
C09976=1113.967,55.698,-54.766,179.952,7.371,149.395
C09977=1113.961,55.947,-54.783,179.952,7.375,149.396
C09978=1113.956,56.196,-54.800,179.953,7.379,149.397
C09979=1113.952,56.446,-54.817,179.955,7.383,149.397
C09980=1113.946,56.695,-54.834,179.956,7.387,149.398
C09981=1113.942,56.945,-54.850,179.957,7.391,149.398
C09982=1113.937,57.193,-54.868,179.958,7.395,149.399
C09983=1113.932,57.443,-54.885,179.960,7.399,149.399
C09984=1113.927,57.692,-54.901,179.960,7.403,149.400
C09985=1113.922,57.942,-54.919,179.962,7.407,149.400
C09986=1113.917,58.191,-54.935,179.963,7.411,149.401
C09987=1113.912,58.441,-54.952,179.965,7.415,149.401
C09988=1113.907,58.690,-54.969,179.966,7.419,149.402
C09989=1113.902,58.940,-54.986,179.967,7.423,149.402
C09990=1113.897,59.189,-55.003,179.969,7.427,149.403
C09991=1113.892,59.438,-55.021,179.969,7.430,149.404
C09992=1113.887,59.687,-55.037,179.971,7.434,149.404
C09993=1113.883,59.937,-55.054,179.972,7.439,149.405
C09994=1113.878,60.186,-55.071,179.974,7.443,149.405
C09995=1113.873,60.436,-55.088,179.975,7.447,149.406
C09996=1113.868,60.685,-55.106,179.976,7.451,149.406
//INST
///DATE 2021/06/25 14:33
///ATTR SC,RW,RJ
////FRAME ROBOT
///GROUP1 RB1
NOP
MOVL C00000 V=800.0 PL=0
MOVL C00001 V=800.0 PL=0
MOVL C00002 V=800.0 PL=0
MOVL C00003 V=800.0 PL=0
MOVL C00004 V=800.0 PL=0
MOVL C00005 V=800.0 PL=0
MOVL C00006 V=800.0 PL=0
MOVL C00007 V=800.0 PL=0
MOVL C00008 V=800.0 PL=0
MOVL C00009 V=800.0 PL=0
MOVL C00010 V=800.0 PL=0
MOVL C00011 V=800.0 PL=0
MOVL C00012 V=800.0 PL=0
MOVL C00013 V=800.0 PL=0
MOVL C00014 V=800.0 PL=0
MOVL C00015 V=800.0 PL=0
MOVL C00016 V=800.0 PL=0
MOVL C00017 V=800.0 PL=0
MOVL C00018 V=800.0 PL=0
MOVL C00019 V=800.0 PL=0
MOVL C00020 V=800.0 PL=0
MOVL C00021 V=800.0 PL=0
MOVL C00022 V=800.0 PL=0
MOVL C00023 V=800.0 PL=0
MOVL C00024 V=800.0 PL=0
MOVL C00025 V=800.0 PL=0
MOVL C00026 V=800.0 PL=0
MOVL C00027 V=800.0 PL=0
MOVL C00028 V=800.0 PL=0
MOVL C00029 V=800.0 PL=0
MOVL C00030 V=800.0 PL=0
MOVL C00031 V=800.0 PL=0
MOVL C00032 V=800.0 PL=0
MOVL C00033 V=800.0 PL=0
MOVL C00034 V=800.0 PL=0
MOVL C00035 V=800.0 PL=0
MOVL C00036 V=800.0 PL=0
MOVL C00037 V=800.0 PL=0
MOVL C00038 V=800.0 PL=0
MOVL C00039 V=800.0 PL=0
MOVL C00040 V=800.0 PL=0
MOVL C00041 V=800.0 PL=0
MOVL C00042 V=800.0 PL=0
MOVL C00043 V=800.0 PL=0
MOVL C00044 V=800.0 PL=0
MOVL C00045 V=800.0 PL=0
MOVL C00046 V=800.0 PL=0
MOVL C00047 V=800.0 PL=0
MOVL C00048 V=800.0 PL=0
MOVL C00049 V=800.0 PL=0
MOVL C00050 V=800.0 PL=0
MOVL C00051 V=800.0 PL=0
MOVL C00052 V=800.0 PL=0
MOVL C00053 V=800.0 PL=0
MOVL C00054 V=800.0 PL=0
MOVL C00055 V=800.0 PL=0
MOVL C00056 V=800.0 PL=0
MOVL C00057 V=800.0 PL=0
MOVL C00058 V=800.0 PL=0
MOVL C00059 V=800.0 PL=0
MOVL C00060 V=800.0 PL=0
MOVL C00061 V=800.0 PL=0
MOVL C00062 V=800.0 PL=0
MOVL C00063 V=800.0 PL=0
MOVL C00064 V=800.0 PL=0
MOVL C00065 V=800.0 PL=0
MOVL C00066 V=800.0 PL=0
MOVL C00067 V=800.0 PL=0
MOVL C00068 V=800.0 PL=0
MOVL C00069 V=800.0 PL=0
MOVL C00070 V=800.0 PL=0
MOVL C00071 V=800.0 PL=0
MOVL C00072 V=800.0 PL=0
MOVL C00073 V=800.0 PL=0
MOVL C00074 V=800.0 PL=0
MOVL C00075 V=800.0 PL=0
MOVL C00076 V=800.0 PL=0
MOVL C00077 V=800.0 PL=0
MOVL C00078 V=800.0 PL=0
MOVL C00079 V=800.0 PL=0
MOVL C00080 V=800.0 PL=0
MOVL C00081 V=800.0 PL=0
MOVL C00082 V=800.0 PL=0
MOVL C00083 V=800.0 PL=0
MOVL C00084 V=800.0 PL=0
MOVL C00085 V=800.0 PL=0
MOVL C00086 V=800.0 PL=0
MOVL C00087 V=800.0 PL=0
MOVL C00088 V=800.0 PL=0
MOVL C00089 V=800.0 PL=0
MOVL C00090 V=800.0 PL=0
MOVL C00091 V=800.0 PL=0
MOVL C00092 V=800.0 PL=0
MOVL C00093 V=800.0 PL=0
MOVL C00094 V=800.0 PL=0
MOVL C00095 V=800.0 PL=0
MOVL C00096 V=800.0 PL=0
MOVL C00097 V=800.0 PL=0
MOVL C00098 V=800.0 PL=0
MOVL C00099 V=800.0 PL=0
MOVL C00100 V=800.0 PL=0
MOVL C00101 V=800.0 PL=0
MOVL C00102 V=800.0 PL=0
MOVL C00103 V=800.0 PL=0
MOVL C00104 V=800.0 PL=0
MOVL C00105 V=800.0 PL=0
MOVL C00106 V=800.0 PL=0
MOVL C00107 V=800.0 PL=0
MOVL C00108 V=800.0 PL=0
MOVL C00109 V=800.0 PL=0
MOVL C00110 V=800.0 PL=0
MOVL C00111 V=800.0 PL=0
MOVL C00112 V=800.0 PL=0
MOVL C00113 V=800.0 PL=0
MOVL C00114 V=800.0 PL=0
MOVL C00115 V=800.0 PL=0
MOVL C00116 V=800.0 PL=0
MOVL C00117 V=800.0 PL=0
MOVL C00118 V=800.0 PL=0
MOVL C00119 V=800.0 PL=0
MOVL C00120 V=800.0 PL=0
MOVL C00121 V=800.0 PL=0
MOVL C00122 V=800.0 PL=0
MOVL C00123 V=800.0 PL=0
MOVL C00124 V=800.0 PL=0
MOVL C00125 V=800.0 PL=0
MOVL C00126 V=800.0 PL=0
MOVL C00127 V=800.0 PL=0
MOVL C00128 V=800.0 PL=0
MOVL C00129 V=800.0 PL=0
MOVL C00130 V=800.0 PL=0
MOVL C00131 V=800.0 PL=0
MOVL C00132 V=800.0 PL=0
MOVL C00133 V=800.0 PL=0
MOVL C00134 V=800.0 PL=0
MOVL C00135 V=800.0 PL=0
MOVL C00136 V=800.0 PL=0
MOVL C00137 V=800.0 PL=0
MOVL C00138 V=800.0 PL=0
MOVL C00139 V=800.0 PL=0
MOVL C00140 V=800.0 PL=0
MOVL C00141 V=800.0 PL=0
MOVL C00142 V=800.0 PL=0
MOVL C00143 V=800.0 PL=0
MOVL C00144 V=800.0 PL=0
MOVL C00145 V=800.0 PL=0
MOVL C00146 V=800.0 PL=0
MOVL C00147 V=800.0 PL=0
MOVL C00148 V=800.0 PL=0
MOVL C00149 V=800.0 PL=0
MOVL C00150 V=800.0 PL=0
MOVL C00151 V=800.0 PL=0
MOVL C00152 V=800.0 PL=0
MOVL C00153 V=800.0 PL=0
MOVL C00154 V=800.0 PL=0
MOVL C00155 V=800.0 PL=0
MOVL C00156 V=800.0 PL=0
MOVL C00157 V=800.0 PL=0
MOVL C00158 V=800.0 PL=0
MOVL C00159 V=800.0 PL=0
MOVL C00160 V=800.0 PL=0
MOVL C00161 V=800.0 PL=0
MOVL C00162 V=800.0 PL=0
MOVL C00163 V=800.0 PL=0
MOVL C00164 V=800.0 PL=0
MOVL C00165 V=800.0 PL=0
MOVL C00166 V=800.0 PL=0
MOVL C00167 V=800.0 PL=0
MOVL C00168 V=800.0 PL=0
MOVL C00169 V=800.0 PL=0
MOVL C00170 V=800.0 PL=0
MOVL C00171 V=800.0 PL=0
MOVL C00172 V=800.0 PL=0
MOVL C00173 V=800.0 PL=0
MOVL C00174 V=800.0 PL=0
MOVL C00175 V=800.0 PL=0
MOVL C00176 V=800.0 PL=0
MOVL C00177 V=800.0 PL=0
MOVL C00178 V=800.0 PL=0
MOVL C00179 V=800.0 PL=0
MOVL C00180 V=800.0 PL=0
MOVL C00181 V=800.0 PL=0
MOVL C00182 V=800.0 PL=0
MOVL C00183 V=800.0 PL=0
MOVL C00184 V=800.0 PL=0
MOVL C00185 V=800.0 PL=0
MOVL C00186 V=800.0 PL=0
MOVL C00187 V=800.0 PL=0
MOVL C00188 V=800.0 PL=0
MOVL C00189 V=800.0 PL=0
MOVL C00190 V=800.0 PL=0
MOVL C00191 V=800.0 PL=0
MOVL C00192 V=800.0 PL=0
MOVL C00193 V=800.0 PL=0
MOVL C00194 V=800.0 PL=0
MOVL C00195 V=800.0 PL=0
MOVL C00196 V=800.0 PL=0
MOVL C00197 V=800.0 PL=0
MOVL C00198 V=800.0 PL=0
MOVL C00199 V=800.0 PL=0
MOVL C00200 V=800.0 PL=0
MOVL C00201 V=800.0 PL=0
MOVL C00202 V=800.0 PL=0
MOVL C00203 V=800.0 PL=0
MOVL C00204 V=800.0 PL=0
MOVL C00205 V=800.0 PL=0
MOVL C00206 V=800.0 PL=0
MOVL C00207 V=800.0 PL=0
MOVL C00208 V=800.0 PL=0
MOVL C00209 V=800.0 PL=0
MOVL C00210 V=800.0 PL=0
MOVL C00211 V=800.0 PL=0
MOVL C00212 V=800.0 PL=0
MOVL C00213 V=800.0 PL=0
MOVL C00214 V=800.0 PL=0
MOVL C00215 V=800.0 PL=0
MOVL C00216 V=800.0 PL=0
MOVL C00217 V=800.0 PL=0
MOVL C00218 V=800.0 PL=0
MOVL C00219 V=800.0 PL=0
MOVL C00220 V=800.0 PL=0
MOVL C00221 V=800.0 PL=0
MOVL C00222 V=800.0 PL=0
MOVL C00223 V=800.0 PL=0
MOVL C00224 V=800.0 PL=0
MOVL C00225 V=800.0 PL=0
MOVL C00226 V=800.0 PL=0
MOVL C00227 V=800.0 PL=0
MOVL C00228 V=800.0 PL=0
MOVL C00229 V=800.0 PL=0
MOVL C00230 V=800.0 PL=0
MOVL C00231 V=800.0 PL=0
MOVL C00232 V=800.0 PL=0
MOVL C00233 V=800.0 PL=0
MOVL C00234 V=800.0 PL=0
MOVL C00235 V=800.0 PL=0
MOVL C00236 V=800.0 PL=0
MOVL C00237 V=800.0 PL=0
MOVL C00238 V=800.0 PL=0
MOVL C00239 V=800.0 PL=0
MOVL C00240 V=800.0 PL=0
MOVL C00241 V=800.0 PL=0
MOVL C00242 V=800.0 PL=0
MOVL C00243 V=800.0 PL=0
MOVL C00244 V=800.0 PL=0
MOVL C00245 V=800.0 PL=0
MOVL C00246 V=800.0 PL=0
MOVL C00247 V=800.0 PL=0
MOVL C00248 V=800.0 PL=0
MOVL C00249 V=800.0 PL=0
MOVL C00250 V=800.0 PL=0
MOVL C00251 V=800.0 PL=0
MOVL C00252 V=800.0 PL=0
MOVL C00253 V=800.0 PL=0
MOVL C00254 V=800.0 PL=0
MOVL C00255 V=800.0 PL=0
MOVL C00256 V=800.0 PL=0
MOVL C00257 V=800.0 PL=0
MOVL C00258 V=800.0 PL=0
MOVL C00259 V=800.0 PL=0
MOVL C00260 V=800.0 PL=0
MOVL C00261 V=800.0 PL=0
MOVL C00262 V=800.0 PL=0
MOVL C00263 V=800.0 PL=0
MOVL C00264 V=800.0 PL=0
MOVL C00265 V=800.0 PL=0
MOVL C00266 V=800.0 PL=0
MOVL C00267 V=800.0 PL=0
MOVL C00268 V=800.0 PL=0
MOVL C00269 V=800.0 PL=0
MOVL C00270 V=800.0 PL=0
MOVL C00271 V=800.0 PL=0
MOVL C00272 V=800.0 PL=0
MOVL C00273 V=800.0 PL=0
MOVL C00274 V=800.0 PL=0
MOVL C00275 V=800.0 PL=0
MOVL C00276 V=800.0 PL=0
MOVL C00277 V=800.0 PL=0
MOVL C00278 V=800.0 PL=0
MOVL C00279 V=800.0 PL=0
MOVL C00280 V=800.0 PL=0
MOVL C00281 V=800.0 PL=0
MOVL C00282 V=800.0 PL=0
MOVL C00283 V=800.0 PL=0
MOVL C00284 V=800.0 PL=0
MOVL C00285 V=800.0 PL=0
MOVL C00286 V=800.0 PL=0
MOVL C00287 V=800.0 PL=0
MOVL C00288 V=800.0 PL=0
MOVL C00289 V=800.0 PL=0
MOVL C00290 V=800.0 PL=0
MOVL C00291 V=800.0 PL=0
MOVL C00292 V=800.0 PL=0
MOVL C00293 V=800.0 PL=0
MOVL C00294 V=800.0 PL=0
MOVL C00295 V=800.0 PL=0
MOVL C00296 V=800.0 PL=0
MOVL C00297 V=800.0 PL=0
MOVL C00298 V=800.0 PL=0
MOVL C00299 V=800.0 PL=0
MOVL C00300 V=800.0 PL=0
MOVL C00301 V=800.0 PL=0
MOVL C00302 V=800.0 PL=0
MOVL C00303 V=800.0 PL=0
MOVL C00304 V=800.0 PL=0
MOVL C00305 V=800.0 PL=0
MOVL C00306 V=800.0 PL=0
MOVL C00307 V=800.0 PL=0
MOVL C00308 V=800.0 PL=0
MOVL C00309 V=800.0 PL=0
MOVL C00310 V=800.0 PL=0
MOVL C00311 V=800.0 PL=0
MOVL C00312 V=800.0 PL=0
MOVL C00313 V=800.0 PL=0
MOVL C00314 V=800.0 PL=0
MOVL C00315 V=800.0 PL=0
MOVL C00316 V=800.0 PL=0
MOVL C00317 V=800.0 PL=0
MOVL C00318 V=800.0 PL=0
MOVL C00319 V=800.0 PL=0
MOVL C00320 V=800.0 PL=0
MOVL C00321 V=800.0 PL=0
MOVL C00322 V=800.0 PL=0
MOVL C00323 V=800.0 PL=0
MOVL C00324 V=800.0 PL=0
MOVL C00325 V=800.0 PL=0
MOVL C00326 V=800.0 PL=0
MOVL C00327 V=800.0 PL=0
MOVL C00328 V=800.0 PL=0
MOVL C00329 V=800.0 PL=0
MOVL C00330 V=800.0 PL=0
MOVL C00331 V=800.0 PL=0
MOVL C00332 V=800.0 PL=0
MOVL C00333 V=800.0 PL=0
MOVL C00334 V=800.0 PL=0
MOVL C00335 V=800.0 PL=0
MOVL C00336 V=800.0 PL=0
MOVL C00337 V=800.0 PL=0
MOVL C00338 V=800.0 PL=0
MOVL C00339 V=800.0 PL=0
MOVL C00340 V=800.0 PL=0
MOVL C00341 V=800.0 PL=0
MOVL C00342 V=800.0 PL=0
MOVL C00343 V=800.0 PL=0
MOVL C00344 V=800.0 PL=0
MOVL C00345 V=800.0 PL=0
MOVL C00346 V=800.0 PL=0
MOVL C00347 V=800.0 PL=0
MOVL C00348 V=800.0 PL=0
MOVL C00349 V=800.0 PL=0
MOVL C00350 V=800.0 PL=0
MOVL C00351 V=800.0 PL=0
MOVL C00352 V=800.0 PL=0
MOVL C00353 V=800.0 PL=0
MOVL C00354 V=800.0 PL=0
MOVL C00355 V=800.0 PL=0
MOVL C00356 V=800.0 PL=0
MOVL C00357 V=800.0 PL=0
MOVL C00358 V=800.0 PL=0
MOVL C00359 V=800.0 PL=0
MOVL C00360 V=800.0 PL=0
MOVL C00361 V=800.0 PL=0
MOVL C00362 V=800.0 PL=0
MOVL C00363 V=800.0 PL=0
MOVL C00364 V=800.0 PL=0
MOVL C00365 V=800.0 PL=0
MOVL C00366 V=800.0 PL=0
MOVL C00367 V=800.0 PL=0
MOVL C00368 V=800.0 PL=0
MOVL C00369 V=800.0 PL=0
MOVL C00370 V=800.0 PL=0
MOVL C00371 V=800.0 PL=0
MOVL C00372 V=800.0 PL=0
MOVL C00373 V=800.0 PL=0
MOVL C00374 V=800.0 PL=0
MOVL C00375 V=800.0 PL=0
MOVL C00376 V=800.0 PL=0
MOVL C00377 V=800.0 PL=0
MOVL C00378 V=800.0 PL=0
MOVL C00379 V=800.0 PL=0
MOVL C00380 V=800.0 PL=0
MOVL C00381 V=800.0 PL=0
MOVL C00382 V=800.0 PL=0
MOVL C00383 V=800.0 PL=0
MOVL C00384 V=800.0 PL=0
MOVL C00385 V=800.0 PL=0
MOVL C00386 V=800.0 PL=0
MOVL C00387 V=800.0 PL=0
MOVL C00388 V=800.0 PL=0
MOVL C00389 V=800.0 PL=0
MOVL C00390 V=800.0 PL=0
MOVL C00391 V=800.0 PL=0
MOVL C00392 V=800.0 PL=0
MOVL C00393 V=800.0 PL=0
MOVL C00394 V=800.0 PL=0
MOVL C00395 V=800.0 PL=0
MOVL C00396 V=800.0 PL=0
MOVL C00397 V=800.0 PL=0
MOVL C00398 V=800.0 PL=0
MOVL C00399 V=800.0 PL=0
MOVL C00400 V=800.0 PL=0
MOVL C00401 V=800.0 PL=0
MOVL C00402 V=800.0 PL=0
MOVL C00403 V=800.0 PL=0
MOVL C00404 V=800.0 PL=0
MOVL C00405 V=800.0 PL=0
MOVL C00406 V=800.0 PL=0
MOVL C00407 V=800.0 PL=0
MOVL C00408 V=800.0 PL=0
MOVL C00409 V=800.0 PL=0
MOVL C00410 V=800.0 PL=0
MOVL C00411 V=800.0 PL=0
MOVL C00412 V=800.0 PL=0
MOVL C00413 V=800.0 PL=0
MOVL C00414 V=800.0 PL=0
MOVL C00415 V=800.0 PL=0
MOVL C00416 V=800.0 PL=0
MOVL C00417 V=800.0 PL=0
MOVL C00418 V=800.0 PL=0
MOVL C00419 V=800.0 PL=0
MOVL C00420 V=800.0 PL=0
MOVL C00421 V=800.0 PL=0
MOVL C00422 V=800.0 PL=0
MOVL C00423 V=800.0 PL=0
MOVL C00424 V=800.0 PL=0
MOVL C00425 V=800.0 PL=0
MOVL C00426 V=800.0 PL=0
MOVL C00427 V=800.0 PL=0
MOVL C00428 V=800.0 PL=0
MOVL C00429 V=800.0 PL=0
MOVL C00430 V=800.0 PL=0
MOVL C00431 V=800.0 PL=0
MOVL C00432 V=800.0 PL=0
MOVL C00433 V=800.0 PL=0
MOVL C00434 V=800.0 PL=0
MOVL C00435 V=800.0 PL=0
MOVL C00436 V=800.0 PL=0
MOVL C00437 V=800.0 PL=0
MOVL C00438 V=800.0 PL=0
MOVL C00439 V=800.0 PL=0
MOVL C00440 V=800.0 PL=0
MOVL C00441 V=800.0 PL=0
MOVL C00442 V=800.0 PL=0
MOVL C00443 V=800.0 PL=0
MOVL C00444 V=800.0 PL=0
MOVL C00445 V=800.0 PL=0
MOVL C00446 V=800.0 PL=0
MOVL C00447 V=800.0 PL=0
MOVL C00448 V=800.0 PL=0
MOVL C00449 V=800.0 PL=0
MOVL C00450 V=800.0 PL=0
MOVL C00451 V=800.0 PL=0
MOVL C00452 V=800.0 PL=0
MOVL C00453 V=800.0 PL=0
MOVL C00454 V=800.0 PL=0
MOVL C00455 V=800.0 PL=0
MOVL C00456 V=800.0 PL=0
MOVL C00457 V=800.0 PL=0
MOVL C00458 V=800.0 PL=0
MOVL C00459 V=800.0 PL=0
MOVL C00460 V=800.0 PL=0
MOVL C00461 V=800.0 PL=0
MOVL C00462 V=800.0 PL=0
MOVL C00463 V=800.0 PL=0
MOVL C00464 V=800.0 PL=0
MOVL C00465 V=800.0 PL=0
MOVL C00466 V=800.0 PL=0
MOVL C00467 V=800.0 PL=0
MOVL C00468 V=800.0 PL=0
MOVL C00469 V=800.0 PL=0
MOVL C00470 V=800.0 PL=0
MOVL C00471 V=800.0 PL=0
MOVL C00472 V=800.0 PL=0
MOVL C00473 V=800.0 PL=0
MOVL C00474 V=800.0 PL=0
MOVL C00475 V=800.0 PL=0
MOVL C00476 V=800.0 PL=0
MOVL C00477 V=800.0 PL=0
MOVL C00478 V=800.0 PL=0
MOVL C00479 V=800.0 PL=0
MOVL C00480 V=800.0 PL=0
MOVL C00481 V=800.0 PL=0
MOVL C00482 V=800.0 PL=0
MOVL C00483 V=800.0 PL=0
MOVL C00484 V=800.0 PL=0
MOVL C00485 V=800.0 PL=0
MOVL C00486 V=800.0 PL=0
MOVL C00487 V=800.0 PL=0
MOVL C00488 V=800.0 PL=0
MOVL C00489 V=800.0 PL=0
MOVL C00490 V=800.0 PL=0
MOVL C00491 V=800.0 PL=0
MOVL C00492 V=800.0 PL=0
MOVL C00493 V=800.0 PL=0
MOVL C00494 V=800.0 PL=0
MOVL C00495 V=800.0 PL=0
MOVL C00496 V=800.0 PL=0
MOVL C00497 V=800.0 PL=0
MOVL C00498 V=800.0 PL=0
MOVL C00499 V=800.0 PL=0
MOVL C00500 V=800.0 PL=0
MOVL C00501 V=800.0 PL=0
MOVL C00502 V=800.0 PL=0
MOVL C00503 V=800.0 PL=0
MOVL C00504 V=800.0 PL=0
MOVL C00505 V=800.0 PL=0
MOVL C00506 V=800.0 PL=0
MOVL C00507 V=800.0 PL=0
MOVL C00508 V=800.0 PL=0
MOVL C00509 V=800.0 PL=0
MOVL C00510 V=800.0 PL=0
MOVL C00511 V=800.0 PL=0
MOVL C00512 V=800.0 PL=0
MOVL C00513 V=800.0 PL=0
MOVL C00514 V=800.0 PL=0
MOVL C00515 V=800.0 PL=0
MOVL C00516 V=800.0 PL=0
MOVL C00517 V=800.0 PL=0
MOVL C00518 V=800.0 PL=0
MOVL C00519 V=800.0 PL=0
MOVL C00520 V=800.0 PL=0
MOVL C00521 V=800.0 PL=0
MOVL C00522 V=800.0 PL=0
MOVL C00523 V=800.0 PL=0
MOVL C00524 V=800.0 PL=0
MOVL C00525 V=800.0 PL=0
MOVL C00526 V=800.0 PL=0
MOVL C00527 V=800.0 PL=0
MOVL C00528 V=800.0 PL=0
MOVL C00529 V=800.0 PL=0
MOVL C00530 V=800.0 PL=0
MOVL C00531 V=800.0 PL=0
MOVL C00532 V=800.0 PL=0
MOVL C00533 V=800.0 PL=0
MOVL C00534 V=800.0 PL=0
MOVL C00535 V=800.0 PL=0
MOVL C00536 V=800.0 PL=0
MOVL C00537 V=800.0 PL=0
MOVL C00538 V=800.0 PL=0
MOVL C00539 V=800.0 PL=0
MOVL C00540 V=800.0 PL=0
MOVL C00541 V=800.0 PL=0
MOVL C00542 V=800.0 PL=0
MOVL C00543 V=800.0 PL=0
MOVL C00544 V=800.0 PL=0
MOVL C00545 V=800.0 PL=0
MOVL C00546 V=800.0 PL=0
MOVL C00547 V=800.0 PL=0
MOVL C00548 V=800.0 PL=0
MOVL C00549 V=800.0 PL=0
MOVL C00550 V=800.0 PL=0
MOVL C00551 V=800.0 PL=0
MOVL C00552 V=800.0 PL=0
MOVL C00553 V=800.0 PL=0
MOVL C00554 V=800.0 PL=0
MOVL C00555 V=800.0 PL=0
MOVL C00556 V=800.0 PL=0
MOVL C00557 V=800.0 PL=0
MOVL C00558 V=800.0 PL=0
MOVL C00559 V=800.0 PL=0
MOVL C00560 V=800.0 PL=0
MOVL C00561 V=800.0 PL=0
MOVL C00562 V=800.0 PL=0
MOVL C00563 V=800.0 PL=0
MOVL C00564 V=800.0 PL=0
MOVL C00565 V=800.0 PL=0
MOVL C00566 V=800.0 PL=0
MOVL C00567 V=800.0 PL=0
MOVL C00568 V=800.0 PL=0
MOVL C00569 V=800.0 PL=0
MOVL C00570 V=800.0 PL=0
MOVL C00571 V=800.0 PL=0
MOVL C00572 V=800.0 PL=0
MOVL C00573 V=800.0 PL=0
MOVL C00574 V=800.0 PL=0
MOVL C00575 V=800.0 PL=0
MOVL C00576 V=800.0 PL=0
MOVL C00577 V=800.0 PL=0
MOVL C00578 V=800.0 PL=0
MOVL C00579 V=800.0 PL=0
MOVL C00580 V=800.0 PL=0
MOVL C00581 V=800.0 PL=0
MOVL C00582 V=800.0 PL=0
MOVL C00583 V=800.0 PL=0
MOVL C00584 V=800.0 PL=0
MOVL C00585 V=800.0 PL=0
MOVL C00586 V=800.0 PL=0
MOVL C00587 V=800.0 PL=0
MOVL C00588 V=800.0 PL=0
MOVL C00589 V=800.0 PL=0
MOVL C00590 V=800.0 PL=0
MOVL C00591 V=800.0 PL=0
MOVL C00592 V=800.0 PL=0
MOVL C00593 V=800.0 PL=0
MOVL C00594 V=800.0 PL=0
MOVL C00595 V=800.0 PL=0
MOVL C00596 V=800.0 PL=0
MOVL C00597 V=800.0 PL=0
MOVL C00598 V=800.0 PL=0
MOVL C00599 V=800.0 PL=0
MOVL C00600 V=800.0 PL=0
MOVL C00601 V=800.0 PL=0
MOVL C00602 V=800.0 PL=0
MOVL C00603 V=800.0 PL=0
MOVL C00604 V=800.0 PL=0
MOVL C00605 V=800.0 PL=0
MOVL C00606 V=800.0 PL=0
MOVL C00607 V=800.0 PL=0
MOVL C00608 V=800.0 PL=0
MOVL C00609 V=800.0 PL=0
MOVL C00610 V=800.0 PL=0
MOVL C00611 V=800.0 PL=0
MOVL C00612 V=800.0 PL=0
MOVL C00613 V=800.0 PL=0
MOVL C00614 V=800.0 PL=0
MOVL C00615 V=800.0 PL=0
MOVL C00616 V=800.0 PL=0
MOVL C00617 V=800.0 PL=0
MOVL C00618 V=800.0 PL=0
MOVL C00619 V=800.0 PL=0
MOVL C00620 V=800.0 PL=0
MOVL C00621 V=800.0 PL=0
MOVL C00622 V=800.0 PL=0
MOVL C00623 V=800.0 PL=0
MOVL C00624 V=800.0 PL=0
MOVL C00625 V=800.0 PL=0
MOVL C00626 V=800.0 PL=0
MOVL C00627 V=800.0 PL=0
MOVL C00628 V=800.0 PL=0
MOVL C00629 V=800.0 PL=0
MOVL C00630 V=800.0 PL=0
MOVL C00631 V=800.0 PL=0
MOVL C00632 V=800.0 PL=0
MOVL C00633 V=800.0 PL=0
MOVL C00634 V=800.0 PL=0
MOVL C00635 V=800.0 PL=0
MOVL C00636 V=800.0 PL=0
MOVL C00637 V=800.0 PL=0
MOVL C00638 V=800.0 PL=0
MOVL C00639 V=800.0 PL=0
MOVL C00640 V=800.0 PL=0
MOVL C00641 V=800.0 PL=0
MOVL C00642 V=800.0 PL=0
MOVL C00643 V=800.0 PL=0
MOVL C00644 V=800.0 PL=0
MOVL C00645 V=800.0 PL=0
MOVL C00646 V=800.0 PL=0
MOVL C00647 V=800.0 PL=0
MOVL C00648 V=800.0 PL=0
MOVL C00649 V=800.0 PL=0
MOVL C00650 V=800.0 PL=0
MOVL C00651 V=800.0 PL=0
MOVL C00652 V=800.0 PL=0
MOVL C00653 V=800.0 PL=0
MOVL C00654 V=800.0 PL=0
MOVL C00655 V=800.0 PL=0
MOVL C00656 V=800.0 PL=0
MOVL C00657 V=800.0 PL=0
MOVL C00658 V=800.0 PL=0
MOVL C00659 V=800.0 PL=0
MOVL C00660 V=800.0 PL=0
MOVL C00661 V=800.0 PL=0
MOVL C00662 V=800.0 PL=0
MOVL C00663 V=800.0 PL=0
MOVL C00664 V=800.0 PL=0
MOVL C00665 V=800.0 PL=0
MOVL C00666 V=800.0 PL=0
MOVL C00667 V=800.0 PL=0
MOVL C00668 V=800.0 PL=0
MOVL C00669 V=800.0 PL=0
MOVL C00670 V=800.0 PL=0
MOVL C00671 V=800.0 PL=0
MOVL C00672 V=800.0 PL=0
MOVL C00673 V=800.0 PL=0
MOVL C00674 V=800.0 PL=0
MOVL C00675 V=800.0 PL=0
MOVL C00676 V=800.0 PL=0
MOVL C00677 V=800.0 PL=0
MOVL C00678 V=800.0 PL=0
MOVL C00679 V=800.0 PL=0
MOVL C00680 V=800.0 PL=0
MOVL C00681 V=800.0 PL=0
MOVL C00682 V=800.0 PL=0
MOVL C00683 V=800.0 PL=0
MOVL C00684 V=800.0 PL=0
MOVL C00685 V=800.0 PL=0
MOVL C00686 V=800.0 PL=0
MOVL C00687 V=800.0 PL=0
MOVL C00688 V=800.0 PL=0
MOVL C00689 V=800.0 PL=0
MOVL C00690 V=800.0 PL=0
MOVL C00691 V=800.0 PL=0
MOVL C00692 V=800.0 PL=0
MOVL C00693 V=800.0 PL=0
MOVL C00694 V=800.0 PL=0
MOVL C00695 V=800.0 PL=0
MOVL C00696 V=800.0 PL=0
MOVL C00697 V=800.0 PL=0
MOVL C00698 V=800.0 PL=0
MOVL C00699 V=800.0 PL=0
MOVL C00700 V=800.0 PL=0
MOVL C00701 V=800.0 PL=0
MOVL C00702 V=800.0 PL=0
MOVL C00703 V=800.0 PL=0
MOVL C00704 V=800.0 PL=0
MOVL C00705 V=800.0 PL=0
MOVL C00706 V=800.0 PL=0
MOVL C00707 V=800.0 PL=0
MOVL C00708 V=800.0 PL=0
MOVL C00709 V=800.0 PL=0
MOVL C00710 V=800.0 PL=0
MOVL C00711 V=800.0 PL=0
MOVL C00712 V=800.0 PL=0
MOVL C00713 V=800.0 PL=0
MOVL C00714 V=800.0 PL=0
MOVL C00715 V=800.0 PL=0
MOVL C00716 V=800.0 PL=0
MOVL C00717 V=800.0 PL=0
MOVL C00718 V=800.0 PL=0
MOVL C00719 V=800.0 PL=0
MOVL C00720 V=800.0 PL=0
MOVL C00721 V=800.0 PL=0
MOVL C00722 V=800.0 PL=0
MOVL C00723 V=800.0 PL=0
MOVL C00724 V=800.0 PL=0
MOVL C00725 V=800.0 PL=0
MOVL C00726 V=800.0 PL=0
MOVL C00727 V=800.0 PL=0
MOVL C00728 V=800.0 PL=0
MOVL C00729 V=800.0 PL=0
MOVL C00730 V=800.0 PL=0
MOVL C00731 V=800.0 PL=0
MOVL C00732 V=800.0 PL=0
MOVL C00733 V=800.0 PL=0
MOVL C00734 V=800.0 PL=0
MOVL C00735 V=800.0 PL=0
MOVL C00736 V=800.0 PL=0
MOVL C00737 V=800.0 PL=0
MOVL C00738 V=800.0 PL=0
MOVL C00739 V=800.0 PL=0
MOVL C00740 V=800.0 PL=0
MOVL C00741 V=800.0 PL=0
MOVL C00742 V=800.0 PL=0
MOVL C00743 V=800.0 PL=0
MOVL C00744 V=800.0 PL=0
MOVL C00745 V=800.0 PL=0
MOVL C00746 V=800.0 PL=0
MOVL C00747 V=800.0 PL=0
MOVL C00748 V=800.0 PL=0
MOVL C00749 V=800.0 PL=0
MOVL C00750 V=800.0 PL=0
MOVL C00751 V=800.0 PL=0
MOVL C00752 V=800.0 PL=0
MOVL C00753 V=800.0 PL=0
MOVL C00754 V=800.0 PL=0
MOVL C00755 V=800.0 PL=0
MOVL C00756 V=800.0 PL=0
MOVL C00757 V=800.0 PL=0
MOVL C00758 V=800.0 PL=0
MOVL C00759 V=800.0 PL=0
MOVL C00760 V=800.0 PL=0
MOVL C00761 V=800.0 PL=0
MOVL C00762 V=800.0 PL=0
MOVL C00763 V=800.0 PL=0
MOVL C00764 V=800.0 PL=0
MOVL C00765 V=800.0 PL=0
MOVL C00766 V=800.0 PL=0
MOVL C00767 V=800.0 PL=0
MOVL C00768 V=800.0 PL=0
MOVL C00769 V=800.0 PL=0
MOVL C00770 V=800.0 PL=0
MOVL C00771 V=800.0 PL=0
MOVL C00772 V=800.0 PL=0
MOVL C00773 V=800.0 PL=0
MOVL C00774 V=800.0 PL=0
MOVL C00775 V=800.0 PL=0
MOVL C00776 V=800.0 PL=0
MOVL C00777 V=800.0 PL=0
MOVL C00778 V=800.0 PL=0
MOVL C00779 V=800.0 PL=0
MOVL C00780 V=800.0 PL=0
MOVL C00781 V=800.0 PL=0
MOVL C00782 V=800.0 PL=0
MOVL C00783 V=800.0 PL=0
MOVL C00784 V=800.0 PL=0
MOVL C00785 V=800.0 PL=0
MOVL C00786 V=800.0 PL=0
MOVL C00787 V=800.0 PL=0
MOVL C00788 V=800.0 PL=0
MOVL C00789 V=800.0 PL=0
MOVL C00790 V=800.0 PL=0
MOVL C00791 V=800.0 PL=0
MOVL C00792 V=800.0 PL=0
MOVL C00793 V=800.0 PL=0
MOVL C00794 V=800.0 PL=0
MOVL C00795 V=800.0 PL=0
MOVL C00796 V=800.0 PL=0
MOVL C00797 V=800.0 PL=0
MOVL C00798 V=800.0 PL=0
MOVL C00799 V=800.0 PL=0
MOVL C00800 V=800.0 PL=0
MOVL C00801 V=800.0 PL=0
MOVL C00802 V=800.0 PL=0
MOVL C00803 V=800.0 PL=0
MOVL C00804 V=800.0 PL=0
MOVL C00805 V=800.0 PL=0
MOVL C00806 V=800.0 PL=0
MOVL C00807 V=800.0 PL=0
MOVL C00808 V=800.0 PL=0
MOVL C00809 V=800.0 PL=0
MOVL C00810 V=800.0 PL=0
MOVL C00811 V=800.0 PL=0
MOVL C00812 V=800.0 PL=0
MOVL C00813 V=800.0 PL=0
MOVL C00814 V=800.0 PL=0
MOVL C00815 V=800.0 PL=0
MOVL C00816 V=800.0 PL=0
MOVL C00817 V=800.0 PL=0
MOVL C00818 V=800.0 PL=0
MOVL C00819 V=800.0 PL=0
MOVL C00820 V=800.0 PL=0
MOVL C00821 V=800.0 PL=0
MOVL C00822 V=800.0 PL=0
MOVL C00823 V=800.0 PL=0
MOVL C00824 V=800.0 PL=0
MOVL C00825 V=800.0 PL=0
MOVL C00826 V=800.0 PL=0
MOVL C00827 V=800.0 PL=0
MOVL C00828 V=800.0 PL=0
MOVL C00829 V=800.0 PL=0
MOVL C00830 V=800.0 PL=0
MOVL C00831 V=800.0 PL=0
MOVL C00832 V=800.0 PL=0
MOVL C00833 V=800.0 PL=0
MOVL C00834 V=800.0 PL=0
MOVL C00835 V=800.0 PL=0
MOVL C00836 V=800.0 PL=0
MOVL C00837 V=800.0 PL=0
MOVL C00838 V=800.0 PL=0
MOVL C00839 V=800.0 PL=0
MOVL C00840 V=800.0 PL=0
MOVL C00841 V=800.0 PL=0
MOVL C00842 V=800.0 PL=0
MOVL C00843 V=800.0 PL=0
MOVL C00844 V=800.0 PL=0
MOVL C00845 V=800.0 PL=0
MOVL C00846 V=800.0 PL=0
MOVL C00847 V=800.0 PL=0
MOVL C00848 V=800.0 PL=0
MOVL C00849 V=800.0 PL=0
MOVL C00850 V=800.0 PL=0
MOVL C00851 V=800.0 PL=0
MOVL C00852 V=800.0 PL=0
MOVL C00853 V=800.0 PL=0
MOVL C00854 V=800.0 PL=0
MOVL C00855 V=800.0 PL=0
MOVL C00856 V=800.0 PL=0
MOVL C00857 V=800.0 PL=0
MOVL C00858 V=800.0 PL=0
MOVL C00859 V=800.0 PL=0
MOVL C00860 V=800.0 PL=0
MOVL C00861 V=800.0 PL=0
MOVL C00862 V=800.0 PL=0
MOVL C00863 V=800.0 PL=0
MOVL C00864 V=800.0 PL=0
MOVL C00865 V=800.0 PL=0
MOVL C00866 V=800.0 PL=0
MOVL C00867 V=800.0 PL=0
MOVL C00868 V=800.0 PL=0
MOVL C00869 V=800.0 PL=0
MOVL C00870 V=800.0 PL=0
MOVL C00871 V=800.0 PL=0
MOVL C00872 V=800.0 PL=0
MOVL C00873 V=800.0 PL=0
MOVL C00874 V=800.0 PL=0
MOVL C00875 V=800.0 PL=0
MOVL C00876 V=800.0 PL=0
MOVL C00877 V=800.0 PL=0
MOVL C00878 V=800.0 PL=0
MOVL C00879 V=800.0 PL=0
MOVL C00880 V=800.0 PL=0
MOVL C00881 V=800.0 PL=0
MOVL C00882 V=800.0 PL=0
MOVL C00883 V=800.0 PL=0
MOVL C00884 V=800.0 PL=0
MOVL C00885 V=800.0 PL=0
MOVL C00886 V=800.0 PL=0
MOVL C00887 V=800.0 PL=0
MOVL C00888 V=800.0 PL=0
MOVL C00889 V=800.0 PL=0
MOVL C00890 V=800.0 PL=0
MOVL C00891 V=800.0 PL=0
MOVL C00892 V=800.0 PL=0
MOVL C00893 V=800.0 PL=0
MOVL C00894 V=800.0 PL=0
MOVL C00895 V=800.0 PL=0
MOVL C00896 V=800.0 PL=0
MOVL C00897 V=800.0 PL=0
MOVL C00898 V=800.0 PL=0
MOVL C00899 V=800.0 PL=0
MOVL C00900 V=800.0 PL=0
MOVL C00901 V=800.0 PL=0
MOVL C00902 V=800.0 PL=0
MOVL C00903 V=800.0 PL=0
MOVL C00904 V=800.0 PL=0
MOVL C00905 V=800.0 PL=0
MOVL C00906 V=800.0 PL=0
MOVL C00907 V=800.0 PL=0
MOVL C00908 V=800.0 PL=0
MOVL C00909 V=800.0 PL=0
MOVL C00910 V=800.0 PL=0
MOVL C00911 V=800.0 PL=0
MOVL C00912 V=800.0 PL=0
MOVL C00913 V=800.0 PL=0
MOVL C00914 V=800.0 PL=0
MOVL C00915 V=800.0 PL=0
MOVL C00916 V=800.0 PL=0
MOVL C00917 V=800.0 PL=0
MOVL C00918 V=800.0 PL=0
MOVL C00919 V=800.0 PL=0
MOVL C00920 V=800.0 PL=0
MOVL C00921 V=800.0 PL=0
MOVL C00922 V=800.0 PL=0
MOVL C00923 V=800.0 PL=0
MOVL C00924 V=800.0 PL=0
MOVL C00925 V=800.0 PL=0
MOVL C00926 V=800.0 PL=0
MOVL C00927 V=800.0 PL=0
MOVL C00928 V=800.0 PL=0
MOVL C00929 V=800.0 PL=0
MOVL C00930 V=800.0 PL=0
MOVL C00931 V=800.0 PL=0
MOVL C00932 V=800.0 PL=0
MOVL C00933 V=800.0 PL=0
MOVL C00934 V=800.0 PL=0
MOVL C00935 V=800.0 PL=0
MOVL C00936 V=800.0 PL=0
MOVL C00937 V=800.0 PL=0
MOVL C00938 V=800.0 PL=0
MOVL C00939 V=800.0 PL=0
MOVL C00940 V=800.0 PL=0
MOVL C00941 V=800.0 PL=0
MOVL C00942 V=800.0 PL=0
MOVL C00943 V=800.0 PL=0
MOVL C00944 V=800.0 PL=0
MOVL C00945 V=800.0 PL=0
MOVL C00946 V=800.0 PL=0
MOVL C00947 V=800.0 PL=0
MOVL C00948 V=800.0 PL=0
MOVL C00949 V=800.0 PL=0
MOVL C00950 V=800.0 PL=0
MOVL C00951 V=800.0 PL=0
MOVL C00952 V=800.0 PL=0
MOVL C00953 V=800.0 PL=0
MOVL C00954 V=800.0 PL=0
MOVL C00955 V=800.0 PL=0
MOVL C00956 V=800.0 PL=0
MOVL C00957 V=800.0 PL=0
MOVL C00958 V=800.0 PL=0
MOVL C00959 V=800.0 PL=0
MOVL C00960 V=800.0 PL=0
MOVL C00961 V=800.0 PL=0
MOVL C00962 V=800.0 PL=0
MOVL C00963 V=800.0 PL=0
MOVL C00964 V=800.0 PL=0
MOVL C00965 V=800.0 PL=0
MOVL C00966 V=800.0 PL=0
MOVL C00967 V=800.0 PL=0
MOVL C00968 V=800.0 PL=0
MOVL C00969 V=800.0 PL=0
MOVL C00970 V=800.0 PL=0
MOVL C00971 V=800.0 PL=0
MOVL C00972 V=800.0 PL=0
MOVL C00973 V=800.0 PL=0
MOVL C00974 V=800.0 PL=0
MOVL C00975 V=800.0 PL=0
MOVL C00976 V=800.0 PL=0
MOVL C00977 V=800.0 PL=0
MOVL C00978 V=800.0 PL=0
MOVL C00979 V=800.0 PL=0
MOVL C00980 V=800.0 PL=0
MOVL C00981 V=800.0 PL=0
MOVL C00982 V=800.0 PL=0
MOVL C00983 V=800.0 PL=0
MOVL C00984 V=800.0 PL=0
MOVL C00985 V=800.0 PL=0
MOVL C00986 V=800.0 PL=0
MOVL C00987 V=800.0 PL=0
MOVL C00988 V=800.0 PL=0
MOVL C00989 V=800.0 PL=0
MOVL C00990 V=800.0 PL=0
MOVL C00991 V=800.0 PL=0
MOVL C00992 V=800.0 PL=0
MOVL C00993 V=800.0 PL=0
MOVL C00994 V=800.0 PL=0
MOVL C00995 V=800.0 PL=0
MOVL C00996 V=800.0 PL=0
MOVL C00997 V=800.0 PL=0
MOVL C00998 V=800.0 PL=0
MOVL C00999 V=800.0 PL=0
MOVL C01000 V=800.0 PL=0
MOVL C01001 V=800.0 PL=0
MOVL C01002 V=800.0 PL=0
MOVL C01003 V=800.0 PL=0
MOVL C01004 V=800.0 PL=0
MOVL C01005 V=800.0 PL=0
MOVL C01006 V=800.0 PL=0
MOVL C01007 V=800.0 PL=0
MOVL C01008 V=800.0 PL=0
MOVL C01009 V=800.0 PL=0
MOVL C01010 V=800.0 PL=0
MOVL C01011 V=800.0 PL=0
MOVL C01012 V=800.0 PL=0
MOVL C01013 V=800.0 PL=0
MOVL C01014 V=800.0 PL=0
MOVL C01015 V=800.0 PL=0
MOVL C01016 V=800.0 PL=0
MOVL C01017 V=800.0 PL=0
MOVL C01018 V=800.0 PL=0
MOVL C01019 V=800.0 PL=0
MOVL C01020 V=800.0 PL=0
MOVL C01021 V=800.0 PL=0
MOVL C01022 V=800.0 PL=0
MOVL C01023 V=800.0 PL=0
MOVL C01024 V=800.0 PL=0
MOVL C01025 V=800.0 PL=0
MOVL C01026 V=800.0 PL=0
MOVL C01027 V=800.0 PL=0
MOVL C01028 V=800.0 PL=0
MOVL C01029 V=800.0 PL=0
MOVL C01030 V=800.0 PL=0
MOVL C01031 V=800.0 PL=0
MOVL C01032 V=800.0 PL=0
MOVL C01033 V=800.0 PL=0
MOVL C01034 V=800.0 PL=0
MOVL C01035 V=800.0 PL=0
MOVL C01036 V=800.0 PL=0
MOVL C01037 V=800.0 PL=0
MOVL C01038 V=800.0 PL=0
MOVL C01039 V=800.0 PL=0
MOVL C01040 V=800.0 PL=0
MOVL C01041 V=800.0 PL=0
MOVL C01042 V=800.0 PL=0
MOVL C01043 V=800.0 PL=0
MOVL C01044 V=800.0 PL=0
MOVL C01045 V=800.0 PL=0
MOVL C01046 V=800.0 PL=0
MOVL C01047 V=800.0 PL=0
MOVL C01048 V=800.0 PL=0
MOVL C01049 V=800.0 PL=0
MOVL C01050 V=800.0 PL=0
MOVL C01051 V=800.0 PL=0
MOVL C01052 V=800.0 PL=0
MOVL C01053 V=800.0 PL=0
MOVL C01054 V=800.0 PL=0
MOVL C01055 V=800.0 PL=0
MOVL C01056 V=800.0 PL=0
MOVL C01057 V=800.0 PL=0
MOVL C01058 V=800.0 PL=0
MOVL C01059 V=800.0 PL=0
MOVL C01060 V=800.0 PL=0
MOVL C01061 V=800.0 PL=0
MOVL C01062 V=800.0 PL=0
MOVL C01063 V=800.0 PL=0
MOVL C01064 V=800.0 PL=0
MOVL C01065 V=800.0 PL=0
MOVL C01066 V=800.0 PL=0
MOVL C01067 V=800.0 PL=0
MOVL C01068 V=800.0 PL=0
MOVL C01069 V=800.0 PL=0
MOVL C01070 V=800.0 PL=0
MOVL C01071 V=800.0 PL=0
MOVL C01072 V=800.0 PL=0
MOVL C01073 V=800.0 PL=0
MOVL C01074 V=800.0 PL=0
MOVL C01075 V=800.0 PL=0
MOVL C01076 V=800.0 PL=0
MOVL C01077 V=800.0 PL=0
MOVL C01078 V=800.0 PL=0
MOVL C01079 V=800.0 PL=0
MOVL C01080 V=800.0 PL=0
MOVL C01081 V=800.0 PL=0
MOVL C01082 V=800.0 PL=0
MOVL C01083 V=800.0 PL=0
MOVL C01084 V=800.0 PL=0
MOVL C01085 V=800.0 PL=0
MOVL C01086 V=800.0 PL=0
MOVL C01087 V=800.0 PL=0
MOVL C01088 V=800.0 PL=0
MOVL C01089 V=800.0 PL=0
MOVL C01090 V=800.0 PL=0
MOVL C01091 V=800.0 PL=0
MOVL C01092 V=800.0 PL=0
MOVL C01093 V=800.0 PL=0
MOVL C01094 V=800.0 PL=0
MOVL C01095 V=800.0 PL=0
MOVL C01096 V=800.0 PL=0
MOVL C01097 V=800.0 PL=0
MOVL C01098 V=800.0 PL=0
MOVL C01099 V=800.0 PL=0
MOVL C01100 V=800.0 PL=0
MOVL C01101 V=800.0 PL=0
MOVL C01102 V=800.0 PL=0
MOVL C01103 V=800.0 PL=0
MOVL C01104 V=800.0 PL=0
MOVL C01105 V=800.0 PL=0
MOVL C01106 V=800.0 PL=0
MOVL C01107 V=800.0 PL=0
MOVL C01108 V=800.0 PL=0
MOVL C01109 V=800.0 PL=0
MOVL C01110 V=800.0 PL=0
MOVL C01111 V=800.0 PL=0
MOVL C01112 V=800.0 PL=0
MOVL C01113 V=800.0 PL=0
MOVL C01114 V=800.0 PL=0
MOVL C01115 V=800.0 PL=0
MOVL C01116 V=800.0 PL=0
MOVL C01117 V=800.0 PL=0
MOVL C01118 V=800.0 PL=0
MOVL C01119 V=800.0 PL=0
MOVL C01120 V=800.0 PL=0
MOVL C01121 V=800.0 PL=0
MOVL C01122 V=800.0 PL=0
MOVL C01123 V=800.0 PL=0
MOVL C01124 V=800.0 PL=0
MOVL C01125 V=800.0 PL=0
MOVL C01126 V=800.0 PL=0
MOVL C01127 V=800.0 PL=0
MOVL C01128 V=800.0 PL=0
MOVL C01129 V=800.0 PL=0
MOVL C01130 V=800.0 PL=0
MOVL C01131 V=800.0 PL=0
MOVL C01132 V=800.0 PL=0
MOVL C01133 V=800.0 PL=0
MOVL C01134 V=800.0 PL=0
MOVL C01135 V=800.0 PL=0
MOVL C01136 V=800.0 PL=0
MOVL C01137 V=800.0 PL=0
MOVL C01138 V=800.0 PL=0
MOVL C01139 V=800.0 PL=0
MOVL C01140 V=800.0 PL=0
MOVL C01141 V=800.0 PL=0
MOVL C01142 V=800.0 PL=0
MOVL C01143 V=800.0 PL=0
MOVL C01144 V=800.0 PL=0
MOVL C01145 V=800.0 PL=0
MOVL C01146 V=800.0 PL=0
MOVL C01147 V=800.0 PL=0
MOVL C01148 V=800.0 PL=0
MOVL C01149 V=800.0 PL=0
MOVL C01150 V=800.0 PL=0
MOVL C01151 V=800.0 PL=0
MOVL C01152 V=800.0 PL=0
MOVL C01153 V=800.0 PL=0
MOVL C01154 V=800.0 PL=0
MOVL C01155 V=800.0 PL=0
MOVL C01156 V=800.0 PL=0
MOVL C01157 V=800.0 PL=0
MOVL C01158 V=800.0 PL=0
MOVL C01159 V=800.0 PL=0
MOVL C01160 V=800.0 PL=0
MOVL C01161 V=800.0 PL=0
MOVL C01162 V=800.0 PL=0
MOVL C01163 V=800.0 PL=0
MOVL C01164 V=800.0 PL=0
MOVL C01165 V=800.0 PL=0
MOVL C01166 V=800.0 PL=0
MOVL C01167 V=800.0 PL=0
MOVL C01168 V=800.0 PL=0
MOVL C01169 V=800.0 PL=0
MOVL C01170 V=800.0 PL=0
MOVL C01171 V=800.0 PL=0
MOVL C01172 V=800.0 PL=0
MOVL C01173 V=800.0 PL=0
MOVL C01174 V=800.0 PL=0
MOVL C01175 V=800.0 PL=0
MOVL C01176 V=800.0 PL=0
MOVL C01177 V=800.0 PL=0
MOVL C01178 V=800.0 PL=0
MOVL C01179 V=800.0 PL=0
MOVL C01180 V=800.0 PL=0
MOVL C01181 V=800.0 PL=0
MOVL C01182 V=800.0 PL=0
MOVL C01183 V=800.0 PL=0
MOVL C01184 V=800.0 PL=0
MOVL C01185 V=800.0 PL=0
MOVL C01186 V=800.0 PL=0
MOVL C01187 V=800.0 PL=0
MOVL C01188 V=800.0 PL=0
MOVL C01189 V=800.0 PL=0
MOVL C01190 V=800.0 PL=0
MOVL C01191 V=800.0 PL=0
MOVL C01192 V=800.0 PL=0
MOVL C01193 V=800.0 PL=0
MOVL C01194 V=800.0 PL=0
MOVL C01195 V=800.0 PL=0
MOVL C01196 V=800.0 PL=0
MOVL C01197 V=800.0 PL=0
MOVL C01198 V=800.0 PL=0
MOVL C01199 V=800.0 PL=0
MOVL C01200 V=800.0 PL=0
MOVL C01201 V=800.0 PL=0
MOVL C01202 V=800.0 PL=0
MOVL C01203 V=800.0 PL=0
MOVL C01204 V=800.0 PL=0
MOVL C01205 V=800.0 PL=0
MOVL C01206 V=800.0 PL=0
MOVL C01207 V=800.0 PL=0
MOVL C01208 V=800.0 PL=0
MOVL C01209 V=800.0 PL=0
MOVL C01210 V=800.0 PL=0
MOVL C01211 V=800.0 PL=0
MOVL C01212 V=800.0 PL=0
MOVL C01213 V=800.0 PL=0
MOVL C01214 V=800.0 PL=0
MOVL C01215 V=800.0 PL=0
MOVL C01216 V=800.0 PL=0
MOVL C01217 V=800.0 PL=0
MOVL C01218 V=800.0 PL=0
MOVL C01219 V=800.0 PL=0
MOVL C01220 V=800.0 PL=0
MOVL C01221 V=800.0 PL=0
MOVL C01222 V=800.0 PL=0
MOVL C01223 V=800.0 PL=0
MOVL C01224 V=800.0 PL=0
MOVL C01225 V=800.0 PL=0
MOVL C01226 V=800.0 PL=0
MOVL C01227 V=800.0 PL=0
MOVL C01228 V=800.0 PL=0
MOVL C01229 V=800.0 PL=0
MOVL C01230 V=800.0 PL=0
MOVL C01231 V=800.0 PL=0
MOVL C01232 V=800.0 PL=0
MOVL C01233 V=800.0 PL=0
MOVL C01234 V=800.0 PL=0
MOVL C01235 V=800.0 PL=0
MOVL C01236 V=800.0 PL=0
MOVL C01237 V=800.0 PL=0
MOVL C01238 V=800.0 PL=0
MOVL C01239 V=800.0 PL=0
MOVL C01240 V=800.0 PL=0
MOVL C01241 V=800.0 PL=0
MOVL C01242 V=800.0 PL=0
MOVL C01243 V=800.0 PL=0
MOVL C01244 V=800.0 PL=0
MOVL C01245 V=800.0 PL=0
MOVL C01246 V=800.0 PL=0
MOVL C01247 V=800.0 PL=0
MOVL C01248 V=800.0 PL=0
MOVL C01249 V=800.0 PL=0
MOVL C01250 V=800.0 PL=0
MOVL C01251 V=800.0 PL=0
MOVL C01252 V=800.0 PL=0
MOVL C01253 V=800.0 PL=0
MOVL C01254 V=800.0 PL=0
MOVL C01255 V=800.0 PL=0
MOVL C01256 V=800.0 PL=0
MOVL C01257 V=800.0 PL=0
MOVL C01258 V=800.0 PL=0
MOVL C01259 V=800.0 PL=0
MOVL C01260 V=800.0 PL=0
MOVL C01261 V=800.0 PL=0
MOVL C01262 V=800.0 PL=0
MOVL C01263 V=800.0 PL=0
MOVL C01264 V=800.0 PL=0
MOVL C01265 V=800.0 PL=0
MOVL C01266 V=800.0 PL=0
MOVL C01267 V=800.0 PL=0
MOVL C01268 V=800.0 PL=0
MOVL C01269 V=800.0 PL=0
MOVL C01270 V=800.0 PL=0
MOVL C01271 V=800.0 PL=0
MOVL C01272 V=800.0 PL=0
MOVL C01273 V=800.0 PL=0
MOVL C01274 V=800.0 PL=0
MOVL C01275 V=800.0 PL=0
MOVL C01276 V=800.0 PL=0
MOVL C01277 V=800.0 PL=0
MOVL C01278 V=800.0 PL=0
MOVL C01279 V=800.0 PL=0
MOVL C01280 V=800.0 PL=0
MOVL C01281 V=800.0 PL=0
MOVL C01282 V=800.0 PL=0
MOVL C01283 V=800.0 PL=0
MOVL C01284 V=800.0 PL=0
MOVL C01285 V=800.0 PL=0
MOVL C01286 V=800.0 PL=0
MOVL C01287 V=800.0 PL=0
MOVL C01288 V=800.0 PL=0
MOVL C01289 V=800.0 PL=0
MOVL C01290 V=800.0 PL=0
MOVL C01291 V=800.0 PL=0
MOVL C01292 V=800.0 PL=0
MOVL C01293 V=800.0 PL=0
MOVL C01294 V=800.0 PL=0
MOVL C01295 V=800.0 PL=0
MOVL C01296 V=800.0 PL=0
MOVL C01297 V=800.0 PL=0
MOVL C01298 V=800.0 PL=0
MOVL C01299 V=800.0 PL=0
MOVL C01300 V=800.0 PL=0
MOVL C01301 V=800.0 PL=0
MOVL C01302 V=800.0 PL=0
MOVL C01303 V=800.0 PL=0
MOVL C01304 V=800.0 PL=0
MOVL C01305 V=800.0 PL=0
MOVL C01306 V=800.0 PL=0
MOVL C01307 V=800.0 PL=0
MOVL C01308 V=800.0 PL=0
MOVL C01309 V=800.0 PL=0
MOVL C01310 V=800.0 PL=0
MOVL C01311 V=800.0 PL=0
MOVL C01312 V=800.0 PL=0
MOVL C01313 V=800.0 PL=0
MOVL C01314 V=800.0 PL=0
MOVL C01315 V=800.0 PL=0
MOVL C01316 V=800.0 PL=0
MOVL C01317 V=800.0 PL=0
MOVL C01318 V=800.0 PL=0
MOVL C01319 V=800.0 PL=0
MOVL C01320 V=800.0 PL=0
MOVL C01321 V=800.0 PL=0
MOVL C01322 V=800.0 PL=0
MOVL C01323 V=800.0 PL=0
MOVL C01324 V=800.0 PL=0
MOVL C01325 V=800.0 PL=0
MOVL C01326 V=800.0 PL=0
MOVL C01327 V=800.0 PL=0
MOVL C01328 V=800.0 PL=0
MOVL C01329 V=800.0 PL=0
MOVL C01330 V=800.0 PL=0
MOVL C01331 V=800.0 PL=0
MOVL C01332 V=800.0 PL=0
MOVL C01333 V=800.0 PL=0
MOVL C01334 V=800.0 PL=0
MOVL C01335 V=800.0 PL=0
MOVL C01336 V=800.0 PL=0
MOVL C01337 V=800.0 PL=0
MOVL C01338 V=800.0 PL=0
MOVL C01339 V=800.0 PL=0
MOVL C01340 V=800.0 PL=0
MOVL C01341 V=800.0 PL=0
MOVL C01342 V=800.0 PL=0
MOVL C01343 V=800.0 PL=0
MOVL C01344 V=800.0 PL=0
MOVL C01345 V=800.0 PL=0
MOVL C01346 V=800.0 PL=0
MOVL C01347 V=800.0 PL=0
MOVL C01348 V=800.0 PL=0
MOVL C01349 V=800.0 PL=0
MOVL C01350 V=800.0 PL=0
MOVL C01351 V=800.0 PL=0
MOVL C01352 V=800.0 PL=0
MOVL C01353 V=800.0 PL=0
MOVL C01354 V=800.0 PL=0
MOVL C01355 V=800.0 PL=0
MOVL C01356 V=800.0 PL=0
MOVL C01357 V=800.0 PL=0
MOVL C01358 V=800.0 PL=0
MOVL C01359 V=800.0 PL=0
MOVL C01360 V=800.0 PL=0
MOVL C01361 V=800.0 PL=0
MOVL C01362 V=800.0 PL=0
MOVL C01363 V=800.0 PL=0
MOVL C01364 V=800.0 PL=0
MOVL C01365 V=800.0 PL=0
MOVL C01366 V=800.0 PL=0
MOVL C01367 V=800.0 PL=0
MOVL C01368 V=800.0 PL=0
MOVL C01369 V=800.0 PL=0
MOVL C01370 V=800.0 PL=0
MOVL C01371 V=800.0 PL=0
MOVL C01372 V=800.0 PL=0
MOVL C01373 V=800.0 PL=0
MOVL C01374 V=800.0 PL=0
MOVL C01375 V=800.0 PL=0
MOVL C01376 V=800.0 PL=0
MOVL C01377 V=800.0 PL=0
MOVL C01378 V=800.0 PL=0
MOVL C01379 V=800.0 PL=0
MOVL C01380 V=800.0 PL=0
MOVL C01381 V=800.0 PL=0
MOVL C01382 V=800.0 PL=0
MOVL C01383 V=800.0 PL=0
MOVL C01384 V=800.0 PL=0
MOVL C01385 V=800.0 PL=0
MOVL C01386 V=800.0 PL=0
MOVL C01387 V=800.0 PL=0
MOVL C01388 V=800.0 PL=0
MOVL C01389 V=800.0 PL=0
MOVL C01390 V=800.0 PL=0
MOVL C01391 V=800.0 PL=0
MOVL C01392 V=800.0 PL=0
MOVL C01393 V=800.0 PL=0
MOVL C01394 V=800.0 PL=0
MOVL C01395 V=800.0 PL=0
MOVL C01396 V=800.0 PL=0
MOVL C01397 V=800.0 PL=0
MOVL C01398 V=800.0 PL=0
MOVL C01399 V=800.0 PL=0
MOVL C01400 V=800.0 PL=0
MOVL C01401 V=800.0 PL=0
MOVL C01402 V=800.0 PL=0
MOVL C01403 V=800.0 PL=0
MOVL C01404 V=800.0 PL=0
MOVL C01405 V=800.0 PL=0
MOVL C01406 V=800.0 PL=0
MOVL C01407 V=800.0 PL=0
MOVL C01408 V=800.0 PL=0
MOVL C01409 V=800.0 PL=0
MOVL C01410 V=800.0 PL=0
MOVL C01411 V=800.0 PL=0
MOVL C01412 V=800.0 PL=0
MOVL C01413 V=800.0 PL=0
MOVL C01414 V=800.0 PL=0
MOVL C01415 V=800.0 PL=0
MOVL C01416 V=800.0 PL=0
MOVL C01417 V=800.0 PL=0
MOVL C01418 V=800.0 PL=0
MOVL C01419 V=800.0 PL=0
MOVL C01420 V=800.0 PL=0
MOVL C01421 V=800.0 PL=0
MOVL C01422 V=800.0 PL=0
MOVL C01423 V=800.0 PL=0
MOVL C01424 V=800.0 PL=0
MOVL C01425 V=800.0 PL=0
MOVL C01426 V=800.0 PL=0
MOVL C01427 V=800.0 PL=0
MOVL C01428 V=800.0 PL=0
MOVL C01429 V=800.0 PL=0
MOVL C01430 V=800.0 PL=0
MOVL C01431 V=800.0 PL=0
MOVL C01432 V=800.0 PL=0
MOVL C01433 V=800.0 PL=0
MOVL C01434 V=800.0 PL=0
MOVL C01435 V=800.0 PL=0
MOVL C01436 V=800.0 PL=0
MOVL C01437 V=800.0 PL=0
MOVL C01438 V=800.0 PL=0
MOVL C01439 V=800.0 PL=0
MOVL C01440 V=800.0 PL=0
MOVL C01441 V=800.0 PL=0
MOVL C01442 V=800.0 PL=0
MOVL C01443 V=800.0 PL=0
MOVL C01444 V=800.0 PL=0
MOVL C01445 V=800.0 PL=0
MOVL C01446 V=800.0 PL=0
MOVL C01447 V=800.0 PL=0
MOVL C01448 V=800.0 PL=0
MOVL C01449 V=800.0 PL=0
MOVL C01450 V=800.0 PL=0
MOVL C01451 V=800.0 PL=0
MOVL C01452 V=800.0 PL=0
MOVL C01453 V=800.0 PL=0
MOVL C01454 V=800.0 PL=0
MOVL C01455 V=800.0 PL=0
MOVL C01456 V=800.0 PL=0
MOVL C01457 V=800.0 PL=0
MOVL C01458 V=800.0 PL=0
MOVL C01459 V=800.0 PL=0
MOVL C01460 V=800.0 PL=0
MOVL C01461 V=800.0 PL=0
MOVL C01462 V=800.0 PL=0
MOVL C01463 V=800.0 PL=0
MOVL C01464 V=800.0 PL=0
MOVL C01465 V=800.0 PL=0
MOVL C01466 V=800.0 PL=0
MOVL C01467 V=800.0 PL=0
MOVL C01468 V=800.0 PL=0
MOVL C01469 V=800.0 PL=0
MOVL C01470 V=800.0 PL=0
MOVL C01471 V=800.0 PL=0
MOVL C01472 V=800.0 PL=0
MOVL C01473 V=800.0 PL=0
MOVL C01474 V=800.0 PL=0
MOVL C01475 V=800.0 PL=0
MOVL C01476 V=800.0 PL=0
MOVL C01477 V=800.0 PL=0
MOVL C01478 V=800.0 PL=0
MOVL C01479 V=800.0 PL=0
MOVL C01480 V=800.0 PL=0
MOVL C01481 V=800.0 PL=0
MOVL C01482 V=800.0 PL=0
MOVL C01483 V=800.0 PL=0
MOVL C01484 V=800.0 PL=0
MOVL C01485 V=800.0 PL=0
MOVL C01486 V=800.0 PL=0
MOVL C01487 V=800.0 PL=0
MOVL C01488 V=800.0 PL=0
MOVL C01489 V=800.0 PL=0
MOVL C01490 V=800.0 PL=0
MOVL C01491 V=800.0 PL=0
MOVL C01492 V=800.0 PL=0
MOVL C01493 V=800.0 PL=0
MOVL C01494 V=800.0 PL=0
MOVL C01495 V=800.0 PL=0
MOVL C01496 V=800.0 PL=0
MOVL C01497 V=800.0 PL=0
MOVL C01498 V=800.0 PL=0
MOVL C01499 V=800.0 PL=0
MOVL C01500 V=800.0 PL=0
MOVL C01501 V=800.0 PL=0
MOVL C01502 V=800.0 PL=0
MOVL C01503 V=800.0 PL=0
MOVL C01504 V=800.0 PL=0
MOVL C01505 V=800.0 PL=0
MOVL C01506 V=800.0 PL=0
MOVL C01507 V=800.0 PL=0
MOVL C01508 V=800.0 PL=0
MOVL C01509 V=800.0 PL=0
MOVL C01510 V=800.0 PL=0
MOVL C01511 V=800.0 PL=0
MOVL C01512 V=800.0 PL=0
MOVL C01513 V=800.0 PL=0
MOVL C01514 V=800.0 PL=0
MOVL C01515 V=800.0 PL=0
MOVL C01516 V=800.0 PL=0
MOVL C01517 V=800.0 PL=0
MOVL C01518 V=800.0 PL=0
MOVL C01519 V=800.0 PL=0
MOVL C01520 V=800.0 PL=0
MOVL C01521 V=800.0 PL=0
MOVL C01522 V=800.0 PL=0
MOVL C01523 V=800.0 PL=0
MOVL C01524 V=800.0 PL=0
MOVL C01525 V=800.0 PL=0
MOVL C01526 V=800.0 PL=0
MOVL C01527 V=800.0 PL=0
MOVL C01528 V=800.0 PL=0
MOVL C01529 V=800.0 PL=0
MOVL C01530 V=800.0 PL=0
MOVL C01531 V=800.0 PL=0
MOVL C01532 V=800.0 PL=0
MOVL C01533 V=800.0 PL=0
MOVL C01534 V=800.0 PL=0
MOVL C01535 V=800.0 PL=0
MOVL C01536 V=800.0 PL=0
MOVL C01537 V=800.0 PL=0
MOVL C01538 V=800.0 PL=0
MOVL C01539 V=800.0 PL=0
MOVL C01540 V=800.0 PL=0
MOVL C01541 V=800.0 PL=0
MOVL C01542 V=800.0 PL=0
MOVL C01543 V=800.0 PL=0
MOVL C01544 V=800.0 PL=0
MOVL C01545 V=800.0 PL=0
MOVL C01546 V=800.0 PL=0
MOVL C01547 V=800.0 PL=0
MOVL C01548 V=800.0 PL=0
MOVL C01549 V=800.0 PL=0
MOVL C01550 V=800.0 PL=0
MOVL C01551 V=800.0 PL=0
MOVL C01552 V=800.0 PL=0
MOVL C01553 V=800.0 PL=0
MOVL C01554 V=800.0 PL=0
MOVL C01555 V=800.0 PL=0
MOVL C01556 V=800.0 PL=0
MOVL C01557 V=800.0 PL=0
MOVL C01558 V=800.0 PL=0
MOVL C01559 V=800.0 PL=0
MOVL C01560 V=800.0 PL=0
MOVL C01561 V=800.0 PL=0
MOVL C01562 V=800.0 PL=0
MOVL C01563 V=800.0 PL=0
MOVL C01564 V=800.0 PL=0
MOVL C01565 V=800.0 PL=0
MOVL C01566 V=800.0 PL=0
MOVL C01567 V=800.0 PL=0
MOVL C01568 V=800.0 PL=0
MOVL C01569 V=800.0 PL=0
MOVL C01570 V=800.0 PL=0
MOVL C01571 V=800.0 PL=0
MOVL C01572 V=800.0 PL=0
MOVL C01573 V=800.0 PL=0
MOVL C01574 V=800.0 PL=0
MOVL C01575 V=800.0 PL=0
MOVL C01576 V=800.0 PL=0
MOVL C01577 V=800.0 PL=0
MOVL C01578 V=800.0 PL=0
MOVL C01579 V=800.0 PL=0
MOVL C01580 V=800.0 PL=0
MOVL C01581 V=800.0 PL=0
MOVL C01582 V=800.0 PL=0
MOVL C01583 V=800.0 PL=0
MOVL C01584 V=800.0 PL=0
MOVL C01585 V=800.0 PL=0
MOVL C01586 V=800.0 PL=0
MOVL C01587 V=800.0 PL=0
MOVL C01588 V=800.0 PL=0
MOVL C01589 V=800.0 PL=0
MOVL C01590 V=800.0 PL=0
MOVL C01591 V=800.0 PL=0
MOVL C01592 V=800.0 PL=0
MOVL C01593 V=800.0 PL=0
MOVL C01594 V=800.0 PL=0
MOVL C01595 V=800.0 PL=0
MOVL C01596 V=800.0 PL=0
MOVL C01597 V=800.0 PL=0
MOVL C01598 V=800.0 PL=0
MOVL C01599 V=800.0 PL=0
MOVL C01600 V=800.0 PL=0
MOVL C01601 V=800.0 PL=0
MOVL C01602 V=800.0 PL=0
MOVL C01603 V=800.0 PL=0
MOVL C01604 V=800.0 PL=0
MOVL C01605 V=800.0 PL=0
MOVL C01606 V=800.0 PL=0
MOVL C01607 V=800.0 PL=0
MOVL C01608 V=800.0 PL=0
MOVL C01609 V=800.0 PL=0
MOVL C01610 V=800.0 PL=0
MOVL C01611 V=800.0 PL=0
MOVL C01612 V=800.0 PL=0
MOVL C01613 V=800.0 PL=0
MOVL C01614 V=800.0 PL=0
MOVL C01615 V=800.0 PL=0
MOVL C01616 V=800.0 PL=0
MOVL C01617 V=800.0 PL=0
MOVL C01618 V=800.0 PL=0
MOVL C01619 V=800.0 PL=0
MOVL C01620 V=800.0 PL=0
MOVL C01621 V=800.0 PL=0
MOVL C01622 V=800.0 PL=0
MOVL C01623 V=800.0 PL=0
MOVL C01624 V=800.0 PL=0
MOVL C01625 V=800.0 PL=0
MOVL C01626 V=800.0 PL=0
MOVL C01627 V=800.0 PL=0
MOVL C01628 V=800.0 PL=0
MOVL C01629 V=800.0 PL=0
MOVL C01630 V=800.0 PL=0
MOVL C01631 V=800.0 PL=0
MOVL C01632 V=800.0 PL=0
MOVL C01633 V=800.0 PL=0
MOVL C01634 V=800.0 PL=0
MOVL C01635 V=800.0 PL=0
MOVL C01636 V=800.0 PL=0
MOVL C01637 V=800.0 PL=0
MOVL C01638 V=800.0 PL=0
MOVL C01639 V=800.0 PL=0
MOVL C01640 V=800.0 PL=0
MOVL C01641 V=800.0 PL=0
MOVL C01642 V=800.0 PL=0
MOVL C01643 V=800.0 PL=0
MOVL C01644 V=800.0 PL=0
MOVL C01645 V=800.0 PL=0
MOVL C01646 V=800.0 PL=0
MOVL C01647 V=800.0 PL=0
MOVL C01648 V=800.0 PL=0
MOVL C01649 V=800.0 PL=0
MOVL C01650 V=800.0 PL=0
MOVL C01651 V=800.0 PL=0
MOVL C01652 V=800.0 PL=0
MOVL C01653 V=800.0 PL=0
MOVL C01654 V=800.0 PL=0
MOVL C01655 V=800.0 PL=0
MOVL C01656 V=800.0 PL=0
MOVL C01657 V=800.0 PL=0
MOVL C01658 V=800.0 PL=0
MOVL C01659 V=800.0 PL=0
MOVL C01660 V=800.0 PL=0
MOVL C01661 V=800.0 PL=0
MOVL C01662 V=800.0 PL=0
MOVL C01663 V=800.0 PL=0
MOVL C01664 V=800.0 PL=0
MOVL C01665 V=800.0 PL=0
MOVL C01666 V=800.0 PL=0
MOVL C01667 V=800.0 PL=0
MOVL C01668 V=800.0 PL=0
MOVL C01669 V=800.0 PL=0
MOVL C01670 V=800.0 PL=0
MOVL C01671 V=800.0 PL=0
MOVL C01672 V=800.0 PL=0
MOVL C01673 V=800.0 PL=0
MOVL C01674 V=800.0 PL=0
MOVL C01675 V=800.0 PL=0
MOVL C01676 V=800.0 PL=0
MOVL C01677 V=800.0 PL=0
MOVL C01678 V=800.0 PL=0
MOVL C01679 V=800.0 PL=0
MOVL C01680 V=800.0 PL=0
MOVL C01681 V=800.0 PL=0
MOVL C01682 V=800.0 PL=0
MOVL C01683 V=800.0 PL=0
MOVL C01684 V=800.0 PL=0
MOVL C01685 V=800.0 PL=0
MOVL C01686 V=800.0 PL=0
MOVL C01687 V=800.0 PL=0
MOVL C01688 V=800.0 PL=0
MOVL C01689 V=800.0 PL=0
MOVL C01690 V=800.0 PL=0
MOVL C01691 V=800.0 PL=0
MOVL C01692 V=800.0 PL=0
MOVL C01693 V=800.0 PL=0
MOVL C01694 V=800.0 PL=0
MOVL C01695 V=800.0 PL=0
MOVL C01696 V=800.0 PL=0
MOVL C01697 V=800.0 PL=0
MOVL C01698 V=800.0 PL=0
MOVL C01699 V=800.0 PL=0
MOVL C01700 V=800.0 PL=0
MOVL C01701 V=800.0 PL=0
MOVL C01702 V=800.0 PL=0
MOVL C01703 V=800.0 PL=0
MOVL C01704 V=800.0 PL=0
MOVL C01705 V=800.0 PL=0
MOVL C01706 V=800.0 PL=0
MOVL C01707 V=800.0 PL=0
MOVL C01708 V=800.0 PL=0
MOVL C01709 V=800.0 PL=0
MOVL C01710 V=800.0 PL=0
MOVL C01711 V=800.0 PL=0
MOVL C01712 V=800.0 PL=0
MOVL C01713 V=800.0 PL=0
MOVL C01714 V=800.0 PL=0
MOVL C01715 V=800.0 PL=0
MOVL C01716 V=800.0 PL=0
MOVL C01717 V=800.0 PL=0
MOVL C01718 V=800.0 PL=0
MOVL C01719 V=800.0 PL=0
MOVL C01720 V=800.0 PL=0
MOVL C01721 V=800.0 PL=0
MOVL C01722 V=800.0 PL=0
MOVL C01723 V=800.0 PL=0
MOVL C01724 V=800.0 PL=0
MOVL C01725 V=800.0 PL=0
MOVL C01726 V=800.0 PL=0
MOVL C01727 V=800.0 PL=0
MOVL C01728 V=800.0 PL=0
MOVL C01729 V=800.0 PL=0
MOVL C01730 V=800.0 PL=0
MOVL C01731 V=800.0 PL=0
MOVL C01732 V=800.0 PL=0
MOVL C01733 V=800.0 PL=0
MOVL C01734 V=800.0 PL=0
MOVL C01735 V=800.0 PL=0
MOVL C01736 V=800.0 PL=0
MOVL C01737 V=800.0 PL=0
MOVL C01738 V=800.0 PL=0
MOVL C01739 V=800.0 PL=0
MOVL C01740 V=800.0 PL=0
MOVL C01741 V=800.0 PL=0
MOVL C01742 V=800.0 PL=0
MOVL C01743 V=800.0 PL=0
MOVL C01744 V=800.0 PL=0
MOVL C01745 V=800.0 PL=0
MOVL C01746 V=800.0 PL=0
MOVL C01747 V=800.0 PL=0
MOVL C01748 V=800.0 PL=0
MOVL C01749 V=800.0 PL=0
MOVL C01750 V=800.0 PL=0
MOVL C01751 V=800.0 PL=0
MOVL C01752 V=800.0 PL=0
MOVL C01753 V=800.0 PL=0
MOVL C01754 V=800.0 PL=0
MOVL C01755 V=800.0 PL=0
MOVL C01756 V=800.0 PL=0
MOVL C01757 V=800.0 PL=0
MOVL C01758 V=800.0 PL=0
MOVL C01759 V=800.0 PL=0
MOVL C01760 V=800.0 PL=0
MOVL C01761 V=800.0 PL=0
MOVL C01762 V=800.0 PL=0
MOVL C01763 V=800.0 PL=0
MOVL C01764 V=800.0 PL=0
MOVL C01765 V=800.0 PL=0
MOVL C01766 V=800.0 PL=0
MOVL C01767 V=800.0 PL=0
MOVL C01768 V=800.0 PL=0
MOVL C01769 V=800.0 PL=0
MOVL C01770 V=800.0 PL=0
MOVL C01771 V=800.0 PL=0
MOVL C01772 V=800.0 PL=0
MOVL C01773 V=800.0 PL=0
MOVL C01774 V=800.0 PL=0
MOVL C01775 V=800.0 PL=0
MOVL C01776 V=800.0 PL=0
MOVL C01777 V=800.0 PL=0
MOVL C01778 V=800.0 PL=0
MOVL C01779 V=800.0 PL=0
MOVL C01780 V=800.0 PL=0
MOVL C01781 V=800.0 PL=0
MOVL C01782 V=800.0 PL=0
MOVL C01783 V=800.0 PL=0
MOVL C01784 V=800.0 PL=0
MOVL C01785 V=800.0 PL=0
MOVL C01786 V=800.0 PL=0
MOVL C01787 V=800.0 PL=0
MOVL C01788 V=800.0 PL=0
MOVL C01789 V=800.0 PL=0
MOVL C01790 V=800.0 PL=0
MOVL C01791 V=800.0 PL=0
MOVL C01792 V=800.0 PL=0
MOVL C01793 V=800.0 PL=0
MOVL C01794 V=800.0 PL=0
MOVL C01795 V=800.0 PL=0
MOVL C01796 V=800.0 PL=0
MOVL C01797 V=800.0 PL=0
MOVL C01798 V=800.0 PL=0
MOVL C01799 V=800.0 PL=0
MOVL C01800 V=800.0 PL=0
MOVL C01801 V=800.0 PL=0
MOVL C01802 V=800.0 PL=0
MOVL C01803 V=800.0 PL=0
MOVL C01804 V=800.0 PL=0
MOVL C01805 V=800.0 PL=0
MOVL C01806 V=800.0 PL=0
MOVL C01807 V=800.0 PL=0
MOVL C01808 V=800.0 PL=0
MOVL C01809 V=800.0 PL=0
MOVL C01810 V=800.0 PL=0
MOVL C01811 V=800.0 PL=0
MOVL C01812 V=800.0 PL=0
MOVL C01813 V=800.0 PL=0
MOVL C01814 V=800.0 PL=0
MOVL C01815 V=800.0 PL=0
MOVL C01816 V=800.0 PL=0
MOVL C01817 V=800.0 PL=0
MOVL C01818 V=800.0 PL=0
MOVL C01819 V=800.0 PL=0
MOVL C01820 V=800.0 PL=0
MOVL C01821 V=800.0 PL=0
MOVL C01822 V=800.0 PL=0
MOVL C01823 V=800.0 PL=0
MOVL C01824 V=800.0 PL=0
MOVL C01825 V=800.0 PL=0
MOVL C01826 V=800.0 PL=0
MOVL C01827 V=800.0 PL=0
MOVL C01828 V=800.0 PL=0
MOVL C01829 V=800.0 PL=0
MOVL C01830 V=800.0 PL=0
MOVL C01831 V=800.0 PL=0
MOVL C01832 V=800.0 PL=0
MOVL C01833 V=800.0 PL=0
MOVL C01834 V=800.0 PL=0
MOVL C01835 V=800.0 PL=0
MOVL C01836 V=800.0 PL=0
MOVL C01837 V=800.0 PL=0
MOVL C01838 V=800.0 PL=0
MOVL C01839 V=800.0 PL=0
MOVL C01840 V=800.0 PL=0
MOVL C01841 V=800.0 PL=0
MOVL C01842 V=800.0 PL=0
MOVL C01843 V=800.0 PL=0
MOVL C01844 V=800.0 PL=0
MOVL C01845 V=800.0 PL=0
MOVL C01846 V=800.0 PL=0
MOVL C01847 V=800.0 PL=0
MOVL C01848 V=800.0 PL=0
MOVL C01849 V=800.0 PL=0
MOVL C01850 V=800.0 PL=0
MOVL C01851 V=800.0 PL=0
MOVL C01852 V=800.0 PL=0
MOVL C01853 V=800.0 PL=0
MOVL C01854 V=800.0 PL=0
MOVL C01855 V=800.0 PL=0
MOVL C01856 V=800.0 PL=0
MOVL C01857 V=800.0 PL=0
MOVL C01858 V=800.0 PL=0
MOVL C01859 V=800.0 PL=0
MOVL C01860 V=800.0 PL=0
MOVL C01861 V=800.0 PL=0
MOVL C01862 V=800.0 PL=0
MOVL C01863 V=800.0 PL=0
MOVL C01864 V=800.0 PL=0
MOVL C01865 V=800.0 PL=0
MOVL C01866 V=800.0 PL=0
MOVL C01867 V=800.0 PL=0
MOVL C01868 V=800.0 PL=0
MOVL C01869 V=800.0 PL=0
MOVL C01870 V=800.0 PL=0
MOVL C01871 V=800.0 PL=0
MOVL C01872 V=800.0 PL=0
MOVL C01873 V=800.0 PL=0
MOVL C01874 V=800.0 PL=0
MOVL C01875 V=800.0 PL=0
MOVL C01876 V=800.0 PL=0
MOVL C01877 V=800.0 PL=0
MOVL C01878 V=800.0 PL=0
MOVL C01879 V=800.0 PL=0
MOVL C01880 V=800.0 PL=0
MOVL C01881 V=800.0 PL=0
MOVL C01882 V=800.0 PL=0
MOVL C01883 V=800.0 PL=0
MOVL C01884 V=800.0 PL=0
MOVL C01885 V=800.0 PL=0
MOVL C01886 V=800.0 PL=0
MOVL C01887 V=800.0 PL=0
MOVL C01888 V=800.0 PL=0
MOVL C01889 V=800.0 PL=0
MOVL C01890 V=800.0 PL=0
MOVL C01891 V=800.0 PL=0
MOVL C01892 V=800.0 PL=0
MOVL C01893 V=800.0 PL=0
MOVL C01894 V=800.0 PL=0
MOVL C01895 V=800.0 PL=0
MOVL C01896 V=800.0 PL=0
MOVL C01897 V=800.0 PL=0
MOVL C01898 V=800.0 PL=0
MOVL C01899 V=800.0 PL=0
MOVL C01900 V=800.0 PL=0
MOVL C01901 V=800.0 PL=0
MOVL C01902 V=800.0 PL=0
MOVL C01903 V=800.0 PL=0
MOVL C01904 V=800.0 PL=0
MOVL C01905 V=800.0 PL=0
MOVL C01906 V=800.0 PL=0
MOVL C01907 V=800.0 PL=0
MOVL C01908 V=800.0 PL=0
MOVL C01909 V=800.0 PL=0
MOVL C01910 V=800.0 PL=0
MOVL C01911 V=800.0 PL=0
MOVL C01912 V=800.0 PL=0
MOVL C01913 V=800.0 PL=0
MOVL C01914 V=800.0 PL=0
MOVL C01915 V=800.0 PL=0
MOVL C01916 V=800.0 PL=0
MOVL C01917 V=800.0 PL=0
MOVL C01918 V=800.0 PL=0
MOVL C01919 V=800.0 PL=0
MOVL C01920 V=800.0 PL=0
MOVL C01921 V=800.0 PL=0
MOVL C01922 V=800.0 PL=0
MOVL C01923 V=800.0 PL=0
MOVL C01924 V=800.0 PL=0
MOVL C01925 V=800.0 PL=0
MOVL C01926 V=800.0 PL=0
MOVL C01927 V=800.0 PL=0
MOVL C01928 V=800.0 PL=0
MOVL C01929 V=800.0 PL=0
MOVL C01930 V=800.0 PL=0
MOVL C01931 V=800.0 PL=0
MOVL C01932 V=800.0 PL=0
MOVL C01933 V=800.0 PL=0
MOVL C01934 V=800.0 PL=0
MOVL C01935 V=800.0 PL=0
MOVL C01936 V=800.0 PL=0
MOVL C01937 V=800.0 PL=0
MOVL C01938 V=800.0 PL=0
MOVL C01939 V=800.0 PL=0
MOVL C01940 V=800.0 PL=0
MOVL C01941 V=800.0 PL=0
MOVL C01942 V=800.0 PL=0
MOVL C01943 V=800.0 PL=0
MOVL C01944 V=800.0 PL=0
MOVL C01945 V=800.0 PL=0
MOVL C01946 V=800.0 PL=0
MOVL C01947 V=800.0 PL=0
MOVL C01948 V=800.0 PL=0
MOVL C01949 V=800.0 PL=0
MOVL C01950 V=800.0 PL=0
MOVL C01951 V=800.0 PL=0
MOVL C01952 V=800.0 PL=0
MOVL C01953 V=800.0 PL=0
MOVL C01954 V=800.0 PL=0
MOVL C01955 V=800.0 PL=0
MOVL C01956 V=800.0 PL=0
MOVL C01957 V=800.0 PL=0
MOVL C01958 V=800.0 PL=0
MOVL C01959 V=800.0 PL=0
MOVL C01960 V=800.0 PL=0
MOVL C01961 V=800.0 PL=0
MOVL C01962 V=800.0 PL=0
MOVL C01963 V=800.0 PL=0
MOVL C01964 V=800.0 PL=0
MOVL C01965 V=800.0 PL=0
MOVL C01966 V=800.0 PL=0
MOVL C01967 V=800.0 PL=0
MOVL C01968 V=800.0 PL=0
MOVL C01969 V=800.0 PL=0
MOVL C01970 V=800.0 PL=0
MOVL C01971 V=800.0 PL=0
MOVL C01972 V=800.0 PL=0
MOVL C01973 V=800.0 PL=0
MOVL C01974 V=800.0 PL=0
MOVL C01975 V=800.0 PL=0
MOVL C01976 V=800.0 PL=0
MOVL C01977 V=800.0 PL=0
MOVL C01978 V=800.0 PL=0
MOVL C01979 V=800.0 PL=0
MOVL C01980 V=800.0 PL=0
MOVL C01981 V=800.0 PL=0
MOVL C01982 V=800.0 PL=0
MOVL C01983 V=800.0 PL=0
MOVL C01984 V=800.0 PL=0
MOVL C01985 V=800.0 PL=0
MOVL C01986 V=800.0 PL=0
MOVL C01987 V=800.0 PL=0
MOVL C01988 V=800.0 PL=0
MOVL C01989 V=800.0 PL=0
MOVL C01990 V=800.0 PL=0
MOVL C01991 V=800.0 PL=0
MOVL C01992 V=800.0 PL=0
MOVL C01993 V=800.0 PL=0
MOVL C01994 V=800.0 PL=0
MOVL C01995 V=800.0 PL=0
MOVL C01996 V=800.0 PL=0
MOVL C01997 V=800.0 PL=0
MOVL C01998 V=800.0 PL=0
MOVL C01999 V=800.0 PL=0
MOVL C02000 V=800.0 PL=0
MOVL C02001 V=800.0 PL=0
MOVL C02002 V=800.0 PL=0
MOVL C02003 V=800.0 PL=0
MOVL C02004 V=800.0 PL=0
MOVL C02005 V=800.0 PL=0
MOVL C02006 V=800.0 PL=0
MOVL C02007 V=800.0 PL=0
MOVL C02008 V=800.0 PL=0
MOVL C02009 V=800.0 PL=0
MOVL C02010 V=800.0 PL=0
MOVL C02011 V=800.0 PL=0
MOVL C02012 V=800.0 PL=0
MOVL C02013 V=800.0 PL=0
MOVL C02014 V=800.0 PL=0
MOVL C02015 V=800.0 PL=0
MOVL C02016 V=800.0 PL=0
MOVL C02017 V=800.0 PL=0
MOVL C02018 V=800.0 PL=0
MOVL C02019 V=800.0 PL=0
MOVL C02020 V=800.0 PL=0
MOVL C02021 V=800.0 PL=0
MOVL C02022 V=800.0 PL=0
MOVL C02023 V=800.0 PL=0
MOVL C02024 V=800.0 PL=0
MOVL C02025 V=800.0 PL=0
MOVL C02026 V=800.0 PL=0
MOVL C02027 V=800.0 PL=0
MOVL C02028 V=800.0 PL=0
MOVL C02029 V=800.0 PL=0
MOVL C02030 V=800.0 PL=0
MOVL C02031 V=800.0 PL=0
MOVL C02032 V=800.0 PL=0
MOVL C02033 V=800.0 PL=0
MOVL C02034 V=800.0 PL=0
MOVL C02035 V=800.0 PL=0
MOVL C02036 V=800.0 PL=0
MOVL C02037 V=800.0 PL=0
MOVL C02038 V=800.0 PL=0
MOVL C02039 V=800.0 PL=0
MOVL C02040 V=800.0 PL=0
MOVL C02041 V=800.0 PL=0
MOVL C02042 V=800.0 PL=0
MOVL C02043 V=800.0 PL=0
MOVL C02044 V=800.0 PL=0
MOVL C02045 V=800.0 PL=0
MOVL C02046 V=800.0 PL=0
MOVL C02047 V=800.0 PL=0
MOVL C02048 V=800.0 PL=0
MOVL C02049 V=800.0 PL=0
MOVL C02050 V=800.0 PL=0
MOVL C02051 V=800.0 PL=0
MOVL C02052 V=800.0 PL=0
MOVL C02053 V=800.0 PL=0
MOVL C02054 V=800.0 PL=0
MOVL C02055 V=800.0 PL=0
MOVL C02056 V=800.0 PL=0
MOVL C02057 V=800.0 PL=0
MOVL C02058 V=800.0 PL=0
MOVL C02059 V=800.0 PL=0
MOVL C02060 V=800.0 PL=0
MOVL C02061 V=800.0 PL=0
MOVL C02062 V=800.0 PL=0
MOVL C02063 V=800.0 PL=0
MOVL C02064 V=800.0 PL=0
MOVL C02065 V=800.0 PL=0
MOVL C02066 V=800.0 PL=0
MOVL C02067 V=800.0 PL=0
MOVL C02068 V=800.0 PL=0
MOVL C02069 V=800.0 PL=0
MOVL C02070 V=800.0 PL=0
MOVL C02071 V=800.0 PL=0
MOVL C02072 V=800.0 PL=0
MOVL C02073 V=800.0 PL=0
MOVL C02074 V=800.0 PL=0
MOVL C02075 V=800.0 PL=0
MOVL C02076 V=800.0 PL=0
MOVL C02077 V=800.0 PL=0
MOVL C02078 V=800.0 PL=0
MOVL C02079 V=800.0 PL=0
MOVL C02080 V=800.0 PL=0
MOVL C02081 V=800.0 PL=0
MOVL C02082 V=800.0 PL=0
MOVL C02083 V=800.0 PL=0
MOVL C02084 V=800.0 PL=0
MOVL C02085 V=800.0 PL=0
MOVL C02086 V=800.0 PL=0
MOVL C02087 V=800.0 PL=0
MOVL C02088 V=800.0 PL=0
MOVL C02089 V=800.0 PL=0
MOVL C02090 V=800.0 PL=0
MOVL C02091 V=800.0 PL=0
MOVL C02092 V=800.0 PL=0
MOVL C02093 V=800.0 PL=0
MOVL C02094 V=800.0 PL=0
MOVL C02095 V=800.0 PL=0
MOVL C02096 V=800.0 PL=0
MOVL C02097 V=800.0 PL=0
MOVL C02098 V=800.0 PL=0
MOVL C02099 V=800.0 PL=0
MOVL C02100 V=800.0 PL=0
MOVL C02101 V=800.0 PL=0
MOVL C02102 V=800.0 PL=0
MOVL C02103 V=800.0 PL=0
MOVL C02104 V=800.0 PL=0
MOVL C02105 V=800.0 PL=0
MOVL C02106 V=800.0 PL=0
MOVL C02107 V=800.0 PL=0
MOVL C02108 V=800.0 PL=0
MOVL C02109 V=800.0 PL=0
MOVL C02110 V=800.0 PL=0
MOVL C02111 V=800.0 PL=0
MOVL C02112 V=800.0 PL=0
MOVL C02113 V=800.0 PL=0
MOVL C02114 V=800.0 PL=0
MOVL C02115 V=800.0 PL=0
MOVL C02116 V=800.0 PL=0
MOVL C02117 V=800.0 PL=0
MOVL C02118 V=800.0 PL=0
MOVL C02119 V=800.0 PL=0
MOVL C02120 V=800.0 PL=0
MOVL C02121 V=800.0 PL=0
MOVL C02122 V=800.0 PL=0
MOVL C02123 V=800.0 PL=0
MOVL C02124 V=800.0 PL=0
MOVL C02125 V=800.0 PL=0
MOVL C02126 V=800.0 PL=0
MOVL C02127 V=800.0 PL=0
MOVL C02128 V=800.0 PL=0
MOVL C02129 V=800.0 PL=0
MOVL C02130 V=800.0 PL=0
MOVL C02131 V=800.0 PL=0
MOVL C02132 V=800.0 PL=0
MOVL C02133 V=800.0 PL=0
MOVL C02134 V=800.0 PL=0
MOVL C02135 V=800.0 PL=0
MOVL C02136 V=800.0 PL=0
MOVL C02137 V=800.0 PL=0
MOVL C02138 V=800.0 PL=0
MOVL C02139 V=800.0 PL=0
MOVL C02140 V=800.0 PL=0
MOVL C02141 V=800.0 PL=0
MOVL C02142 V=800.0 PL=0
MOVL C02143 V=800.0 PL=0
MOVL C02144 V=800.0 PL=0
MOVL C02145 V=800.0 PL=0
MOVL C02146 V=800.0 PL=0
MOVL C02147 V=800.0 PL=0
MOVL C02148 V=800.0 PL=0
MOVL C02149 V=800.0 PL=0
MOVL C02150 V=800.0 PL=0
MOVL C02151 V=800.0 PL=0
MOVL C02152 V=800.0 PL=0
MOVL C02153 V=800.0 PL=0
MOVL C02154 V=800.0 PL=0
MOVL C02155 V=800.0 PL=0
MOVL C02156 V=800.0 PL=0
MOVL C02157 V=800.0 PL=0
MOVL C02158 V=800.0 PL=0
MOVL C02159 V=800.0 PL=0
MOVL C02160 V=800.0 PL=0
MOVL C02161 V=800.0 PL=0
MOVL C02162 V=800.0 PL=0
MOVL C02163 V=800.0 PL=0
MOVL C02164 V=800.0 PL=0
MOVL C02165 V=800.0 PL=0
MOVL C02166 V=800.0 PL=0
MOVL C02167 V=800.0 PL=0
MOVL C02168 V=800.0 PL=0
MOVL C02169 V=800.0 PL=0
MOVL C02170 V=800.0 PL=0
MOVL C02171 V=800.0 PL=0
MOVL C02172 V=800.0 PL=0
MOVL C02173 V=800.0 PL=0
MOVL C02174 V=800.0 PL=0
MOVL C02175 V=800.0 PL=0
MOVL C02176 V=800.0 PL=0
MOVL C02177 V=800.0 PL=0
MOVL C02178 V=800.0 PL=0
